C05376=1015.693,102.871,-118.305,166.533,55.921,160.218
C05377=1015.698,103.121,-118.324,166.535,55.912,160.217
C05378=1015.703,103.370,-118.340,166.538,55.902,160.216
C05379=1015.707,103.620,-118.357,166.541,55.892,160.214
C05380=1015.712,103.869,-118.375,166.544,55.882,160.213
C05381=1015.717,104.119,-118.392,166.546,55.872,160.212
C05382=1015.721,104.368,-118.409,166.549,55.862,160.210
C05383=1015.726,104.617,-118.427,166.551,55.852,160.209
C05384=1015.730,104.866,-118.444,166.555,55.842,160.208
C05385=1015.735,105.115,-118.462,166.558,55.832,160.206
C05386=1015.740,105.365,-118.479,166.560,55.822,160.205
C05387=1015.745,105.614,-118.496,166.563,55.812,160.204
C05388=1015.753,106.033,-118.526,166.567,55.795,160.202
C05389=1015.761,106.451,-118.554,166.572,55.778,160.199
C05390=1015.768,106.870,-118.583,166.577,55.761,160.197
C05391=1015.777,107.288,-118.612,166.582,55.744,160.195
C05392=1015.781,107.538,-118.630,166.584,55.735,160.194
C05393=1015.786,107.787,-118.647,166.587,55.724,160.192
C05394=1015.791,108.037,-118.665,166.590,55.714,160.191
C05395=1015.796,108.286,-118.682,166.593,55.704,160.190
C05396=1015.800,108.535,-118.699,166.596,55.694,160.188
C05397=1015.806,108.784,-118.717,166.598,55.684,160.187
C05398=1015.810,109.034,-118.734,166.601,55.673,160.185
C05399=1015.814,109.283,-118.751,166.605,55.664,160.184
C05400=1015.820,109.532,-118.769,166.607,55.654,160.183
C05401=1015.825,109.782,-118.787,166.610,55.644,160.182
C05402=1015.829,110.032,-118.804,166.612,55.634,160.180
C05403=1015.833,110.280,-118.822,166.615,55.623,160.179
C05404=1015.838,110.530,-118.839,166.618,55.614,160.177
C05405=1015.843,110.779,-118.857,166.621,55.604,160.176
C05406=1015.848,111.029,-118.875,166.625,55.594,160.175
C05407=1015.853,111.278,-118.892,166.627,55.584,160.173
C05408=1015.857,111.527,-118.910,166.630,55.573,160.172
C05409=1015.862,111.777,-118.928,166.632,55.564,160.171
C05410=1015.867,112.026,-118.946,166.635,55.554,160.170
C05411=1015.871,112.275,-118.964,166.639,55.544,160.168
C05412=1015.876,112.524,-118.982,166.641,55.534,160.167
C05413=1015.880,112.774,-118.999,166.644,55.525,160.166
C05414=1015.885,113.024,-119.017,166.647,55.514,160.164
C05415=1015.889,113.272,-119.035,166.649,55.505,160.163
C05416=1015.894,113.522,-119.053,166.652,55.495,160.162
C05417=1015.899,113.771,-119.071,166.656,55.485,160.161
C05418=1015.903,114.021,-119.089,166.658,55.475,160.159
C05419=1015.908,114.270,-119.107,166.662,55.465,160.158
C05420=1015.912,114.519,-119.125,166.664,55.455,160.157
C05421=1015.917,114.768,-119.143,166.667,55.445,160.155
C05422=1015.922,115.018,-119.161,166.670,55.435,160.154
C05423=1015.926,115.268,-119.179,166.673,55.425,160.153
C05424=1015.931,115.517,-119.197,166.675,55.416,160.151
C05425=1015.935,115.766,-119.215,166.678,55.405,160.150
C05426=1015.940,116.015,-119.233,166.681,55.396,160.149
C05427=1015.945,116.264,-119.251,166.684,55.386,160.147
C05428=1015.949,116.514,-119.269,166.687,55.376,160.146
C05429=1015.954,116.763,-119.287,166.690,55.366,160.145
C05430=1015.958,117.012,-119.305,166.693,55.356,160.143
C05431=1015.963,117.262,-119.322,166.696,55.346,160.142
C05432=1015.968,117.511,-119.341,166.699,55.336,160.141
C05433=1015.972,117.760,-119.359,166.701,55.327,160.140
C05434=1015.977,118.010,-119.377,166.705,55.316,160.138
C05435=1015.982,118.259,-119.395,166.707,55.307,160.137
C05436=1015.987,118.508,-119.413,166.710,55.297,160.136
C05437=1015.991,118.757,-119.431,166.713,55.286,160.134
C05438=1015.996,119.006,-119.449,166.716,55.277,160.133
C05439=1016.000,119.256,-119.467,166.719,55.266,160.132
C05440=1016.005,119.505,-119.486,166.721,55.256,160.130
C05441=1016.010,119.754,-119.504,166.725,55.247,160.129
C05442=1016.015,120.004,-119.522,166.728,55.236,160.128
C05443=1016.020,120.253,-119.540,166.730,55.226,160.126
C05444=1016.024,120.502,-119.558,166.734,55.217,160.125
C05445=1016.028,120.751,-119.576,166.737,55.206,160.124
C05446=1016.033,121.000,-119.594,166.739,55.196,160.122
C05447=1016.038,121.250,-119.612,166.743,55.187,160.121
C05448=1016.043,121.499,-119.630,166.745,55.177,160.120
C05449=1016.048,121.749,-119.649,166.748,55.166,160.118
C05450=1016.052,121.998,-119.667,166.752,55.157,160.117
C05451=1016.057,122.247,-119.685,166.754,55.147,160.116
C05452=1016.063,122.528,-119.706,166.758,55.135,160.114
C05453=1016.067,122.810,-119.725,166.762,55.124,160.113
C05454=1016.073,123.091,-119.746,166.764,55.113,160.111
C05455=1016.078,123.372,-119.766,166.768,55.101,160.110
C05456=1016.082,123.622,-119.785,166.772,55.092,160.109
C05457=1016.087,123.871,-119.803,166.774,55.082,160.107
C05458=1016.092,124.120,-119.821,166.777,55.071,160.106
C05459=1016.097,124.369,-119.840,166.780,55.061,160.105
C05460=1016.102,124.618,-119.858,166.783,55.052,160.104
C05461=1016.106,124.868,-119.877,166.786,55.042,160.102
C05462=1016.111,125.117,-119.895,166.789,55.031,160.101
C05463=1016.116,125.366,-119.913,166.792,55.021,160.099
C05464=1016.121,125.616,-119.931,166.795,55.012,160.098
C05465=1016.126,125.865,-119.949,166.799,55.001,160.097
C05466=1016.130,126.115,-119.967,166.802,54.991,160.096
C05467=1016.135,126.364,-119.986,166.804,54.981,160.094
C05468=1016.140,126.613,-120.004,166.808,54.971,160.093
C05469=1016.145,126.862,-120.023,166.811,54.961,160.092
C05470=1016.150,127.111,-120.041,166.814,54.951,160.090
C05471=1016.155,127.361,-120.059,166.816,54.941,160.089
C05472=1016.159,127.610,-120.077,166.820,54.930,160.088
C05473=1016.164,127.859,-120.095,166.823,54.921,160.087
C05474=1016.169,128.109,-120.113,166.827,54.911,160.085
C05475=1016.174,128.358,-120.132,166.829,54.901,160.084
C05476=1016.179,128.607,-120.150,166.832,54.890,160.082
C05477=1016.184,128.856,-120.169,166.835,54.880,160.081
C05478=1016.188,129.105,-120.187,166.839,54.870,160.080
C05479=1016.193,129.355,-120.205,166.841,54.860,160.079
C05480=1016.197,129.605,-120.224,166.845,54.850,160.077
C05481=1016.202,129.853,-120.243,166.848,54.840,160.076
C05482=1016.207,130.103,-120.261,166.851,54.831,160.075
C05483=1016.211,130.352,-120.280,166.854,54.820,160.073
C05484=1016.216,130.601,-120.298,166.858,54.811,160.072
C05485=1016.220,130.851,-120.317,166.860,54.801,160.071
C05486=1016.225,131.099,-120.336,166.863,54.791,160.069
C05487=1016.231,131.349,-120.355,166.867,54.781,160.068
C05488=1016.235,131.598,-120.374,166.869,54.771,160.067
C05489=1016.240,131.848,-120.392,166.873,54.761,160.066
C05490=1016.244,132.097,-120.411,166.876,54.751,160.065
C05491=1016.249,132.346,-120.430,166.879,54.741,160.063
C05492=1016.254,132.596,-120.448,166.882,54.731,160.062
C05493=1016.258,132.845,-120.467,166.886,54.721,160.061
C05494=1016.263,133.094,-120.486,166.888,54.712,160.059
C05495=1016.267,133.343,-120.505,166.891,54.701,160.058
C05496=1016.272,133.592,-120.523,166.895,54.692,160.057
C05497=1016.277,133.841,-120.542,166.898,54.681,160.055
C05498=1016.282,134.091,-120.561,166.901,54.672,160.054
C05499=1016.287,134.340,-120.580,166.904,54.662,160.053
C05500=1016.291,134.590,-120.599,166.908,54.652,160.052
C05501=1016.296,134.839,-120.618,166.910,54.642,160.050
C05502=1016.301,135.088,-120.636,166.914,54.632,160.049
C05503=1016.305,135.337,-120.655,166.917,54.622,160.048
C05504=1016.310,135.586,-120.674,166.921,54.612,160.046
C05505=1016.314,135.835,-120.693,166.923,54.602,160.045
C05506=1016.320,136.085,-120.712,166.927,54.592,160.044
C05507=1016.324,136.334,-120.731,166.930,54.582,160.043
C05508=1016.329,136.583,-120.750,166.932,54.572,160.041
C05509=1016.333,136.833,-120.769,166.936,54.563,160.040
C05510=1016.338,137.082,-120.788,166.939,54.552,160.039
C05511=1016.342,137.331,-120.806,166.943,54.542,160.037
C05512=1016.348,137.581,-120.826,166.946,54.533,160.036
C05513=1016.352,137.830,-120.845,166.949,54.523,160.035
C05514=1016.357,138.079,-120.863,166.952,54.512,160.034
C05515=1016.361,138.328,-120.883,166.955,54.503,160.032
C05516=1016.366,138.609,-120.905,166.959,54.492,160.031
C05517=1016.372,138.890,-120.926,166.963,54.481,160.030
C05518=1016.377,139.171,-120.947,166.966,54.470,160.028
C05519=1016.382,139.452,-120.969,166.970,54.458,160.027
C05520=1016.387,139.702,-120.989,166.974,54.449,160.026
C05521=1016.392,139.951,-121.007,166.977,54.439,160.024
C05522=1016.396,140.200,-121.027,166.980,54.429,160.023
C05523=1016.400,140.449,-121.046,166.983,54.419,160.022
C05524=1016.406,140.699,-121.065,166.986,54.409,160.020
C05525=1016.410,140.948,-121.085,166.989,54.400,160.019
C05526=1016.415,141.197,-121.104,166.993,54.390,160.018
C05527=1016.420,141.446,-121.122,166.996,54.379,160.017
C05528=1016.424,141.695,-121.142,167.000,54.370,160.016
C05529=1016.429,141.945,-121.162,167.002,54.360,160.014
C05530=1016.434,142.194,-121.181,167.006,54.350,160.013
C05531=1016.438,142.443,-121.200,167.010,54.340,160.012
C05532=1016.442,142.692,-121.219,167.013,54.330,160.010
C05533=1016.448,142.942,-121.238,167.015,54.320,160.009
C05534=1016.452,143.191,-121.258,167.019,54.311,160.008
C05535=1016.457,143.440,-121.277,167.023,54.301,160.007
C05536=1016.462,143.689,-121.296,167.026,54.290,160.005
C05537=1016.467,143.938,-121.316,167.029,54.281,160.004
C05538=1016.471,144.187,-121.335,167.032,54.271,160.003
C05539=1016.476,144.436,-121.354,167.036,54.261,160.001
C05540=1016.481,144.686,-121.374,167.040,54.251,160.000
C05541=1016.485,144.935,-121.393,167.043,54.241,159.999
C05542=1016.490,145.184,-121.412,167.045,54.231,159.998
C05543=1016.495,145.434,-121.431,167.049,54.222,159.997
C05544=1016.500,145.683,-121.451,167.053,54.212,159.995
C05545=1016.504,145.932,-121.470,167.056,54.202,159.994
C05546=1016.509,146.182,-121.490,167.059,54.192,159.993
C05547=1016.514,146.430,-121.509,167.062,54.182,159.991
C05548=1016.518,146.680,-121.528,167.066,54.173,159.990
C05549=1016.523,146.928,-121.549,167.070,54.163,159.989
C05550=1016.528,147.178,-121.569,167.072,54.153,159.988
C05551=1016.532,147.427,-121.588,167.076,54.143,159.987
C05552=1016.537,147.676,-121.608,167.080,54.133,159.985
C05553=1016.542,147.926,-121.627,167.083,54.124,159.984
C05554=1016.546,148.175,-121.647,167.086,54.114,159.983
C05555=1016.552,148.424,-121.666,167.089,54.104,159.982
C05556=1016.556,148.673,-121.685,167.093,54.094,159.980
C05557=1016.560,148.922,-121.705,167.097,54.084,159.979
C05558=1016.566,149.171,-121.726,167.100,54.075,159.978
C05559=1016.570,149.420,-121.745,167.103,54.065,159.977
C05560=1016.574,149.669,-121.764,167.107,54.055,159.975
C05561=1016.579,149.919,-121.784,167.110,54.045,159.974
C05562=1016.584,150.168,-121.804,167.113,54.035,159.973
C05563=1016.589,150.418,-121.824,167.117,54.026,159.972
C05564=1016.593,150.666,-121.844,167.120,54.016,159.971
C05565=1016.598,150.915,-121.863,167.124,54.006,159.969
C05566=1016.602,151.165,-121.883,167.128,53.996,159.968
C05567=1016.607,151.414,-121.903,167.130,53.986,159.967
C05568=1016.612,151.663,-121.923,167.134,53.977,159.966
C05569=1016.616,151.912,-121.943,167.138,53.967,159.964
C05570=1016.621,152.161,-121.962,167.141,53.957,159.963
C05571=1016.626,152.411,-121.982,167.145,53.947,159.962
C05572=1016.630,152.659,-122.002,167.148,53.938,159.961
C05573=1016.635,152.909,-122.022,167.152,53.928,159.960
C05574=1016.640,153.158,-122.041,167.155,53.918,159.958
C05575=1016.645,153.407,-122.062,167.159,53.908,159.957
C05576=1016.649,153.656,-122.081,167.162,53.898,159.956
C05577=1016.654,153.906,-122.101,167.165,53.889,159.954
C05578=1016.659,154.155,-122.121,167.169,53.879,159.953
C05579=1016.663,154.404,-122.141,167.172,53.869,159.952
C05580=1016.668,154.685,-122.165,167.177,53.858,159.951
C05581=1016.674,154.966,-122.186,167.181,53.847,159.950
C05582=1016.679,155.247,-122.209,167.184,53.837,159.948
C05583=1016.685,155.528,-122.231,167.188,53.825,159.947
C05584=1016.689,155.778,-122.252,167.192,53.815,159.945
C05585=1016.693,156.026,-122.272,167.196,53.806,159.944
C05586=1016.698,156.276,-122.292,167.199,53.796,159.943
C05587=1016.703,156.524,-122.312,167.203,53.786,159.942
C05588=1016.708,156.774,-122.332,167.206,53.777,159.941
C05589=1016.713,157.022,-122.352,167.210,53.767,159.940
C05590=1016.718,157.272,-122.372,167.213,53.757,159.938
C05591=1016.722,157.521,-122.392,167.217,53.747,159.937
C05592=1016.727,157.770,-122.412,167.221,53.738,159.936
C05593=1016.731,158.019,-122.433,167.224,53.727,159.935
C05594=1016.736,158.269,-122.453,167.227,53.718,159.933
C05595=1016.741,158.517,-122.473,167.231,53.708,159.932
C05596=1016.746,158.767,-122.493,167.235,53.699,159.931
C05597=1016.750,159.016,-122.513,167.238,53.689,159.930
C05598=1016.754,159.265,-122.535,167.241,53.680,159.929
C05599=1016.759,159.514,-122.555,167.245,53.670,159.928
C05600=1016.763,159.764,-122.575,167.249,53.660,159.926
C05601=1016.768,160.012,-122.595,167.253,53.651,159.925
C05602=1016.772,160.261,-122.617,167.256,53.642,159.924
C05603=1016.777,160.511,-122.637,167.260,53.632,159.923
C05604=1016.781,160.759,-122.658,167.264,53.623,159.922
C05605=1016.785,161.009,-122.678,167.268,53.613,159.921
C05606=1016.790,161.258,-122.698,167.270,53.603,159.919
C05607=1016.795,161.507,-122.720,167.274,53.594,159.918
C05608=1016.799,161.756,-122.740,167.278,53.584,159.917
C05609=1016.804,162.005,-122.761,167.282,53.575,159.916
C05610=1016.808,162.255,-122.782,167.285,53.566,159.915
C05611=1016.813,162.504,-122.802,167.288,53.556,159.913
C05612=1016.817,162.753,-122.823,167.292,53.546,159.912
C05613=1016.822,163.001,-122.843,167.297,53.537,159.911
C05614=1016.826,163.251,-122.864,167.299,53.527,159.910
C05615=1016.832,163.500,-122.885,167.303,53.518,159.909
C05616=1016.836,163.749,-122.905,167.307,53.508,159.908
C05617=1016.840,163.998,-122.927,167.311,53.498,159.906
C05618=1016.845,164.247,-122.947,167.315,53.489,159.905
C05619=1016.849,164.496,-122.968,167.317,53.479,159.904
C05620=1016.855,164.745,-122.988,167.321,53.470,159.903
C05621=1016.858,164.994,-123.009,167.325,53.460,159.902
C05622=1016.863,165.244,-123.030,167.329,53.451,159.901
C05623=1016.868,165.493,-123.050,167.333,53.441,159.900
C05624=1016.872,165.742,-123.071,167.337,53.431,159.898
C05625=1016.877,165.991,-123.092,167.340,53.422,159.897
C05626=1016.882,166.240,-123.113,167.343,53.412,159.896
C05627=1016.885,166.489,-123.133,167.348,53.403,159.895
C05628=1016.891,166.738,-123.154,167.352,53.394,159.894
C05629=1016.895,166.988,-123.175,167.355,53.384,159.892
C05630=1016.900,167.236,-123.195,167.359,53.374,159.891
C05631=1016.904,167.486,-123.217,167.362,53.365,159.890
C05632=1016.909,167.735,-123.238,167.366,53.355,159.889
C05633=1016.914,167.984,-123.258,167.370,53.346,159.888
C05634=1016.918,168.233,-123.279,167.374,53.336,159.887
C05635=1016.923,168.482,-123.300,167.378,53.327,159.886
C05636=1016.928,168.731,-123.321,167.381,53.317,159.884
C05637=1016.932,168.979,-123.342,167.386,53.307,159.883
C05638=1016.937,169.229,-123.363,167.390,53.298,159.882
C05639=1016.942,169.478,-123.384,167.393,53.288,159.881
C05640=1016.947,169.727,-123.404,167.396,53.279,159.880
C05641=1016.951,169.976,-123.425,167.400,53.269,159.878
C05642=1016.956,170.225,-123.446,167.404,53.260,159.877
C05643=1016.961,170.474,-123.467,167.408,53.250,159.876
C05644=1016.966,170.755,-123.491,167.412,53.239,159.875
C05645=1016.971,171.036,-123.515,167.417,53.228,159.874
C05646=1016.977,171.317,-123.538,167.421,53.218,159.872
C05647=1016.983,171.597,-123.562,167.426,53.207,159.871
C05648=1016.986,171.846,-123.583,167.429,53.197,159.870
C05649=1016.992,172.095,-123.603,167.433,53.187,159.869
C05650=1016.996,172.345,-123.624,167.438,53.178,159.868
C05651=1017.001,172.594,-123.646,167.441,53.168,159.866
C05652=1017.006,172.843,-123.666,167.445,53.159,159.865
C05653=1017.011,173.092,-123.688,167.449,53.149,159.864
C05654=1017.015,173.340,-123.708,167.453,53.140,159.863
C05655=1017.020,173.590,-123.729,167.457,53.130,159.862
C05656=1017.024,173.839,-123.750,167.461,53.120,159.861
C05657=1017.030,174.088,-123.772,167.465,53.110,159.859
C05658=1017.035,174.337,-123.793,167.469,53.101,159.858
C05659=1017.039,174.587,-123.814,167.473,53.092,159.857
C05660=1017.044,174.836,-123.835,167.477,53.082,159.856
C05661=1017.049,175.084,-123.856,167.481,53.073,159.855
C05662=1017.054,175.333,-123.877,167.484,53.063,159.854
C05663=1017.058,175.582,-123.898,167.489,53.053,159.853
C05664=1017.063,175.831,-123.920,167.492,53.043,159.851
C05665=1017.068,176.080,-123.940,167.496,53.034,159.850
C05666=1017.073,176.330,-123.961,167.500,53.024,159.849
C05667=1017.078,176.579,-123.982,167.504,53.015,159.848
C05668=1017.083,176.828,-124.004,167.508,53.006,159.847
C05669=1017.088,177.077,-124.025,167.512,52.996,159.846
C05670=1017.093,177.326,-124.046,167.516,52.986,159.845
C05671=1017.098,177.575,-124.067,167.520,52.976,159.843
C05672=1017.102,177.825,-124.088,167.524,52.967,159.842
C05673=1017.108,178.073,-124.110,167.528,52.957,159.841
C05674=1017.112,178.323,-124.131,167.532,52.948,159.840
C05675=1017.117,178.571,-124.151,167.536,52.938,159.839
C05676=1017.122,178.820,-124.173,167.540,52.929,159.838
C05677=1017.126,179.069,-124.194,167.544,52.919,159.837
C05678=1017.132,179.318,-124.215,167.548,52.910,159.835
C05679=1017.136,179.567,-124.236,167.553,52.899,159.834
C05680=1017.141,179.816,-124.258,167.557,52.890,159.833
C05681=1017.146,180.065,-124.279,167.561,52.881,159.832
C05682=1017.151,180.315,-124.300,167.565,52.871,159.831
C05683=1017.156,180.563,-124.321,167.569,52.862,159.830
C05684=1017.161,180.812,-124.342,167.573,52.852,159.829
C05685=1017.166,181.062,-124.365,167.577,52.843,159.828
C05686=1017.172,181.311,-124.385,167.581,52.833,159.826
C05687=1017.176,181.560,-124.407,167.585,52.823,159.825
C05688=1017.181,181.809,-124.428,167.590,52.813,159.824
C05689=1017.186,182.058,-124.450,167.594,52.804,159.823
C05690=1017.191,182.307,-124.472,167.597,52.795,159.822
C05691=1017.195,182.556,-124.494,167.601,52.786,159.821
C05692=1017.199,182.806,-124.516,167.605,52.777,159.820
C05693=1017.204,183.054,-124.537,167.610,52.767,159.819
C05694=1017.209,183.303,-124.559,167.614,52.758,159.818
C05695=1017.213,183.552,-124.582,167.618,52.749,159.817
C05696=1017.218,183.801,-124.604,167.622,52.739,159.815
C05697=1017.223,184.050,-124.625,167.626,52.730,159.814
C05698=1017.227,184.299,-124.647,167.630,52.721,159.813
C05699=1017.232,184.548,-124.670,167.635,52.711,159.812
C05700=1017.236,184.797,-124.692,167.639,52.702,159.811
C05701=1017.241,185.045,-124.714,167.643,52.693,159.810
C05702=1017.245,185.295,-124.735,167.647,52.684,159.809
C05703=1017.250,185.544,-124.757,167.651,52.675,159.808
C05704=1017.255,185.794,-124.779,167.655,52.665,159.807
C05705=1017.260,186.042,-124.801,167.659,52.656,159.806
C05706=1017.264,186.292,-124.824,167.664,52.646,159.805
C05707=1017.269,186.540,-124.846,167.668,52.637,159.804
C05708=1017.275,186.820,-124.871,167.673,52.627,159.803
C05709=1017.280,187.101,-124.896,167.677,52.616,159.801
C05710=1017.285,187.381,-124.920,167.682,52.606,159.800
C05711=1017.290,187.662,-124.945,167.687,52.596,159.799
C05712=1017.294,187.910,-124.967,167.691,52.586,159.798
C05713=1017.300,188.160,-124.989,167.695,52.577,159.797
C05714=1017.304,188.409,-125.012,167.699,52.568,159.796
C05715=1017.309,188.658,-125.034,167.703,52.558,159.795
C05716=1017.314,188.906,-125.056,167.708,52.549,159.794
C05717=1017.319,189.155,-125.078,167.712,52.540,159.792
C05718=1017.323,189.404,-125.100,167.716,52.531,159.791
C05719=1017.328,189.654,-125.123,167.721,52.521,159.791
C05720=1017.333,189.902,-125.145,167.726,52.512,159.789
C05721=1017.337,190.152,-125.167,167.730,52.503,159.788
C05722=1017.342,190.400,-125.189,167.734,52.494,159.787
C05723=1017.347,190.649,-125.211,167.738,52.484,159.786
C05724=1017.352,190.899,-125.233,167.742,52.475,159.785
C05725=1017.357,191.147,-125.256,167.746,52.465,159.784
C05726=1017.361,191.396,-125.278,167.751,52.456,159.783
C05727=1017.366,191.645,-125.300,167.755,52.447,159.782
C05728=1017.371,191.895,-125.323,167.759,52.438,159.781
C05729=1017.376,192.143,-125.345,167.765,52.429,159.780
C05730=1017.381,192.392,-125.367,167.769,52.419,159.779
C05731=1017.386,192.640,-125.389,167.773,52.410,159.778
C05732=1017.390,192.890,-125.412,167.777,52.400,159.777
C05733=1017.395,193.139,-125.434,167.781,52.391,159.776
C05734=1017.400,193.387,-125.456,167.786,52.382,159.775
C05735=1017.405,193.637,-125.479,167.790,52.373,159.774
C05736=1017.410,193.886,-125.501,167.795,52.364,159.773
C05737=1017.415,194.135,-125.523,167.799,52.354,159.772
C05738=1017.419,194.383,-125.546,167.804,52.345,159.771
C05739=1017.424,194.633,-125.568,167.808,52.335,159.769
C05740=1017.429,194.882,-125.590,167.812,52.326,159.768
C05741=1017.434,195.130,-125.613,167.816,52.317,159.767
C05742=1017.439,195.380,-125.636,167.822,52.308,159.766
C05743=1017.444,195.628,-125.657,167.826,52.299,159.765
C05744=1017.450,195.877,-125.680,167.830,52.289,159.764
C05745=1017.454,196.126,-125.703,167.834,52.280,159.763
C05746=1017.459,196.375,-125.725,167.839,52.271,159.762
C05747=1017.464,196.624,-125.748,167.844,52.262,159.761
C05748=1017.468,196.873,-125.770,167.848,52.253,159.760
C05749=1017.474,197.121,-125.793,167.852,52.243,159.759
C05750=1017.479,197.371,-125.815,167.857,52.234,159.758
C05751=1017.483,197.620,-125.837,167.862,52.224,159.757
C05752=1017.489,197.869,-125.860,167.866,52.215,159.756
C05753=1017.494,198.118,-125.882,167.871,52.206,159.755
C05754=1017.499,198.367,-125.905,167.875,52.197,159.754
C05755=1017.503,198.616,-125.928,167.880,52.188,159.753
C05756=1017.509,198.864,-125.950,167.885,52.178,159.752
C05757=1017.514,199.114,-125.972,167.889,52.169,159.751
C05758=1017.518,199.362,-125.996,167.893,52.160,159.750
C05759=1017.523,199.612,-126.018,167.899,52.151,159.749
C05760=1017.528,199.860,-126.041,167.903,52.142,159.748
C05761=1017.533,200.109,-126.064,167.907,52.133,159.747
C05762=1017.537,200.358,-126.087,167.912,52.124,159.746
C05763=1017.543,200.607,-126.110,167.916,52.114,159.745
C05764=1017.547,200.856,-126.133,167.920,52.105,159.744
C05765=1017.552,201.104,-126.156,167.926,52.096,159.743
C05766=1017.557,201.354,-126.178,167.930,52.087,159.742
C05767=1017.562,201.602,-126.202,167.935,52.078,159.741
C05768=1017.567,201.852,-126.225,167.939,52.069,159.740
C05769=1017.572,202.100,-126.248,167.943,52.060,159.739
C05770=1017.577,202.349,-126.271,167.949,52.051,159.738
C05771=1017.600,203.593,-126.387,168.432,52.137,159.849
C05772=1017.606,203.828,-126.409,168.436,52.129,159.848
C05773=1017.612,204.063,-126.433,168.440,52.122,159.847
C05774=1017.618,204.298,-126.456,168.443,52.114,159.846
C05775=1017.623,204.534,-126.479,168.447,52.107,159.845
C05776=1017.629,204.769,-126.502,168.450,52.099,159.844
C05777=1017.634,205.003,-126.526,168.454,52.091,159.844
C05778=1017.640,205.238,-126.549,168.458,52.084,159.843
C05779=1017.645,205.473,-126.572,168.462,52.076,159.842
C05780=1017.651,205.722,-126.598,168.466,52.068,159.841
C05781=1017.657,205.970,-126.622,168.470,52.061,159.840
C05782=1017.663,206.219,-126.647,168.474,52.053,159.839
C05783=1017.669,206.468,-126.672,168.477,52.045,159.838
C05784=1017.674,206.716,-126.697,168.481,52.037,159.837
C05785=1017.680,206.966,-126.721,168.485,52.030,159.836
C05786=1017.686,207.214,-126.746,168.490,52.021,159.835
C05787=1017.692,207.463,-126.771,168.494,52.013,159.834
C05788=1017.698,207.712,-126.796,168.498,52.006,159.834
C05789=1017.703,207.960,-126.821,168.501,51.998,159.833
C05790=1017.709,208.209,-126.846,168.505,51.990,159.832
C05791=1017.716,208.458,-126.871,168.509,51.983,159.831
C05792=1017.721,208.706,-126.896,168.513,51.975,159.830
C05793=1017.727,208.955,-126.921,168.517,51.967,159.829
C05794=1017.732,209.204,-126.946,168.521,51.960,159.828
C05795=1017.738,209.452,-126.971,168.525,51.951,159.827
C05796=1017.744,209.701,-126.996,168.530,51.944,159.826
C05797=1017.750,209.950,-127.022,168.533,51.936,159.825
C05798=1017.756,210.198,-127.046,168.537,51.929,159.825
C05799=1017.762,210.447,-127.071,168.541,51.921,159.824
C05800=1017.767,210.696,-127.097,168.545,51.913,159.823
C05801=1017.773,210.944,-127.122,168.549,51.905,159.822
C05802=1017.779,211.193,-127.147,168.553,51.898,159.821
C05803=1017.785,211.442,-127.172,168.557,51.890,159.820
C05804=1017.790,211.690,-127.198,168.561,51.883,159.819
C05805=1017.796,211.939,-127.223,168.565,51.876,159.818
C05806=1017.802,212.187,-127.248,168.569,51.868,159.817
C05807=1017.808,212.436,-127.274,168.573,51.860,159.817
C05808=1017.813,212.685,-127.299,168.577,51.853,159.816
C05809=1017.819,212.934,-127.324,168.581,51.845,159.815
C05810=1017.825,213.182,-127.349,168.585,51.838,159.814
C05811=1017.831,213.431,-127.375,168.589,51.830,159.813
C05812=1017.836,213.679,-127.400,168.593,51.823,159.812
C05813=1017.843,213.928,-127.426,168.597,51.816,159.811
C05814=1017.849,214.177,-127.451,168.601,51.808,159.810
C05815=1017.854,214.426,-127.477,168.605,51.800,159.810
C05816=1017.860,214.674,-127.501,168.609,51.793,159.809
C05817=1017.866,214.923,-127.526,168.613,51.786,159.808
C05818=1017.871,215.172,-127.552,168.617,51.778,159.807
C05819=1017.878,215.421,-127.578,168.621,51.771,159.806
C05820=1017.884,215.669,-127.603,168.625,51.763,159.806
C05821=1017.889,215.917,-127.628,168.630,51.756,159.805
C05822=1017.895,216.166,-127.654,168.633,51.748,159.804
C05823=1017.901,216.415,-127.679,168.636,51.741,159.803
C05824=1017.907,216.663,-127.705,168.641,51.734,159.802
C05825=1017.913,216.912,-127.730,168.645,51.727,159.801
C05826=1017.919,217.161,-127.756,168.648,51.719,159.800
C05827=1017.925,217.410,-127.781,168.653,51.712,159.799
C05828=1017.931,217.658,-127.806,168.657,51.704,159.799
C05829=1017.937,217.906,-127.832,168.661,51.697,159.798
C05830=1017.943,218.155,-127.858,168.665,51.690,159.797
C05831=1017.949,218.403,-127.884,168.669,51.683,159.796
C05832=1017.959,218.817,-127.926,168.675,51.671,159.795
C05833=1017.966,219.179,-127.964,168.681,51.660,159.794
C05834=1017.975,219.540,-128.002,168.687,51.650,159.793
C05835=1017.983,219.901,-128.039,168.693,51.640,159.792
C05836=1017.992,220.263,-128.077,168.699,51.629,159.790
C05837=1017.998,220.512,-128.103,168.704,51.622,159.790
C05838=1018.003,220.760,-128.128,168.708,51.615,159.789
C05839=1018.009,221.009,-128.154,168.712,51.608,159.788
C05840=1018.015,221.257,-128.180,168.716,51.600,159.787
C05841=1018.021,221.506,-128.206,168.719,51.594,159.786
C05842=1018.026,221.755,-128.232,168.723,51.586,159.786
C05843=1018.033,222.003,-128.258,168.728,51.580,159.785
C05844=1018.038,222.252,-128.284,168.732,51.573,159.784
C05845=1018.044,222.500,-128.309,168.736,51.565,159.783
C05846=1018.050,222.749,-128.336,168.741,51.558,159.783
C05847=1018.056,222.997,-128.361,168.744,51.551,159.782
C05848=1018.062,223.246,-128.387,168.748,51.544,159.781
C05849=1018.068,223.495,-128.413,168.753,51.537,159.780
C05850=1018.074,223.743,-128.439,168.757,51.530,159.780
C05851=1018.080,223.992,-128.465,168.761,51.523,159.779
C05852=1018.086,224.240,-128.491,168.765,51.516,159.778
C05853=1018.091,224.489,-128.517,168.769,51.510,159.777
C05854=1018.097,224.738,-128.543,168.773,51.502,159.777
C05855=1018.103,224.986,-128.569,168.777,51.495,159.776
C05856=1018.109,225.235,-128.595,168.781,51.488,159.775
C05857=1018.115,225.483,-128.621,168.786,51.482,159.774
C05858=1018.121,225.732,-128.647,168.789,51.475,159.774
C05859=1018.127,225.980,-128.673,168.793,51.467,159.773
C05860=1018.133,226.229,-128.699,168.798,51.461,159.772
C05861=1018.138,226.478,-128.725,168.802,51.454,159.771
C05862=1018.145,226.726,-128.751,168.806,51.447,159.771
C05863=1018.151,226.974,-128.778,168.810,51.440,159.770
C05864=1018.156,227.223,-128.804,168.814,51.433,159.769
C05865=1018.162,227.471,-128.831,168.819,51.427,159.769
C05866=1018.168,227.720,-128.858,168.822,51.420,159.768
C05867=1018.174,227.969,-128.883,168.827,51.413,159.767
C05868=1018.180,228.218,-128.910,168.831,51.406,159.766
C05869=1018.186,228.466,-128.936,168.836,51.400,159.766
C05870=1018.191,228.715,-128.962,168.839,51.393,159.765
C05871=1018.197,228.963,-128.989,168.843,51.386,159.764
C05872=1018.203,229.212,-129.015,168.848,51.379,159.764
C05873=1018.209,229.460,-129.042,168.851,51.373,159.763
C05874=1018.215,229.709,-129.067,168.856,51.366,159.762
C05875=1018.221,229.957,-129.094,168.860,51.359,159.762
C05876=1018.227,230.205,-129.121,168.865,51.353,159.761
C05877=1018.233,230.454,-129.148,168.868,51.347,159.760
C05878=1018.239,230.703,-129.174,168.873,51.339,159.759
C05879=1018.244,230.951,-129.201,168.877,51.333,159.759
C05880=1018.250,231.199,-129.228,168.881,51.327,159.758
C05881=1018.256,231.448,-129.254,168.885,51.320,159.757
C05882=1018.262,231.697,-129.280,168.890,51.313,159.757
C05883=1018.267,231.945,-129.307,168.893,51.307,159.756
C05884=1018.274,232.194,-129.334,168.898,51.300,159.755
C05885=1018.279,232.443,-129.361,168.902,51.293,159.755
C05886=1018.285,232.691,-129.387,168.906,51.287,159.754
C05887=1018.291,232.939,-129.414,168.911,51.281,159.754
C05888=1018.297,233.188,-129.441,168.914,51.275,159.753
C05889=1018.302,233.416,-129.465,168.919,51.268,159.752
C05890=1018.308,233.644,-129.490,168.922,51.262,159.752
C05891=1018.313,233.872,-129.514,168.926,51.256,159.751
C05892=1018.318,234.101,-129.539,168.930,51.250,159.750
C05893=1018.324,234.329,-129.563,168.934,51.244,159.750
C05894=1018.330,234.558,-129.588,168.937,51.238,159.749
C05895=1018.334,234.786,-129.613,168.941,51.233,159.749
C05896=1018.341,235.014,-129.637,168.945,51.226,159.748
C05897=1018.346,235.262,-129.663,168.950,51.220,159.747
C05898=1018.353,235.511,-129.690,168.954,51.213,159.747
C05899=1018.358,235.760,-129.717,168.958,51.207,159.746
C05900=1018.365,236.007,-129.744,168.963,51.201,159.746
C05901=1018.370,236.256,-129.771,168.966,51.195,159.745
C05902=1018.377,236.505,-129.798,168.971,51.188,159.744
C05903=1018.382,236.753,-129.825,168.976,51.182,159.744
C05904=1018.387,237.002,-129.852,168.979,51.176,159.743
C05905=1018.393,237.250,-129.879,168.984,51.169,159.743
C05906=1018.400,237.499,-129.906,168.988,51.162,159.742
C05907=1018.406,237.747,-129.933,168.992,51.156,159.741
C05908=1018.412,237.995,-129.960,168.997,51.150,159.741
C05909=1018.418,238.244,-129.987,169.000,51.144,159.740
C05910=1018.424,238.493,-130.013,169.005,51.138,159.739
C05911=1018.429,238.741,-130.040,169.010,51.131,159.739
C05912=1018.436,238.990,-130.068,169.013,51.125,159.738
C05913=1018.442,239.238,-130.094,169.018,51.118,159.738
C05914=1018.447,239.487,-130.122,169.022,51.112,159.737
C05915=1018.454,239.735,-130.149,169.026,51.106,159.736
C05916=1018.459,239.983,-130.176,169.030,51.100,159.736
C05917=1018.465,240.231,-130.204,169.035,51.094,159.735
C05918=1018.471,240.481,-130.231,169.039,51.088,159.735
C05919=1018.477,240.729,-130.258,169.043,51.081,159.734
C05920=1018.483,240.978,-130.286,169.047,51.075,159.733
C05921=1018.489,241.226,-130.313,169.052,51.070,159.733
C05922=1018.495,241.474,-130.340,169.056,51.063,159.732
C05923=1018.500,241.723,-130.368,169.061,51.057,159.732
C05924=1018.506,241.971,-130.395,169.064,51.051,159.731
C05925=1018.513,242.220,-130.422,169.069,51.045,159.731
C05926=1018.518,242.468,-130.450,169.074,51.039,159.730
C05927=1018.524,242.716,-130.477,169.078,51.033,159.729
C05928=1018.531,242.965,-130.504,169.083,51.027,159.729
C05929=1018.536,243.213,-130.532,169.086,51.021,159.728
C05930=1018.542,243.462,-130.559,169.091,51.015,159.728
C05931=1018.548,243.710,-130.587,169.095,51.009,159.727
C05932=1018.553,243.958,-130.615,169.099,51.003,159.727
C05933=1018.559,244.207,-130.642,169.104,50.997,159.726
C05934=1018.565,244.455,-130.670,169.107,50.991,159.726
C05935=1018.571,244.704,-130.698,169.113,50.985,159.725
C05936=1018.576,244.952,-130.725,169.117,50.980,159.725
C05937=1018.582,245.201,-130.753,169.121,50.973,159.724
C05938=1018.588,245.449,-130.781,169.125,50.968,159.724
C05939=1018.594,245.697,-130.809,169.130,50.961,159.723
C05940=1018.600,245.945,-130.837,169.134,50.956,159.723
C05941=1018.606,246.195,-130.864,169.138,50.950,159.722
C05942=1018.611,246.443,-130.892,169.143,50.944,159.722
C05943=1018.617,246.691,-130.920,169.147,50.939,159.721
C05944=1018.623,246.939,-130.948,169.152,50.932,159.720
C05945=1018.629,247.188,-130.976,169.156,50.927,159.720
C05946=1018.635,247.436,-131.003,169.160,50.920,159.719
C05947=1018.641,247.685,-131.031,169.164,50.915,159.719
C05948=1018.646,247.933,-131.059,169.169,50.910,159.718
C05949=1018.652,248.158,-131.085,169.173,50.904,159.718
C05950=1018.657,248.383,-131.109,169.177,50.899,159.718
C05951=1018.663,248.608,-131.135,169.181,50.893,159.717
C05952=1018.668,248.833,-131.160,169.185,50.888,159.717
C05953=1018.674,249.058,-131.185,169.189,50.883,159.716
C05954=1018.679,249.283,-131.210,169.192,50.878,159.716
C05955=1018.684,249.507,-131.235,169.196,50.873,159.715
C05956=1018.689,249.733,-131.262,169.201,50.867,159.715
C05957=1018.696,249.981,-131.289,169.205,50.862,159.714
C05958=1018.701,250.229,-131.317,169.210,50.856,159.714
C05959=1018.708,250.478,-131.345,169.214,50.851,159.714
C05960=1018.714,250.726,-131.373,169.218,50.844,159.713
C05961=1018.719,250.974,-131.401,169.223,50.839,159.712
C05962=1018.726,251.223,-131.429,169.228,50.833,159.712
C05963=1018.731,251.471,-131.457,169.232,50.828,159.712
C05964=1018.737,251.720,-131.485,169.236,50.822,159.711
C05965=1018.744,251.968,-131.513,169.240,50.816,159.711
C05966=1018.749,252.216,-131.541,169.245,50.811,159.710
C05967=1018.755,252.465,-131.569,169.250,50.805,159.710
C05968=1018.762,252.713,-131.597,169.254,50.799,159.709
C05969=1018.767,252.961,-131.625,169.259,50.794,159.709
C05970=1018.773,253.210,-131.653,169.263,50.788,159.708
C05971=1018.780,253.459,-131.681,169.267,50.783,159.708
C05972=1018.786,253.706,-131.710,169.272,50.777,159.707
C05973=1018.792,253.954,-131.738,169.276,50.771,159.707
C05974=1018.798,254.203,-131.766,169.281,50.765,159.706
C05975=1018.804,254.452,-131.794,169.285,50.760,159.706
C05976=1018.810,254.700,-131.822,169.290,50.754,159.706
C05977=1018.816,254.948,-131.850,169.294,50.749,159.705
C05978=1018.823,255.197,-131.879,169.298,50.744,159.705
C05979=1018.829,255.445,-131.907,169.303,50.738,159.704
C05980=1018.835,255.693,-131.935,169.307,50.732,159.704
C05981=1018.840,255.942,-131.963,169.313,50.727,159.703
C05982=1018.847,256.190,-131.991,169.317,50.721,159.703
C05983=1018.853,256.438,-132.020,169.322,50.716,159.703
C05984=1018.859,256.687,-132.048,169.326,50.710,159.702
C05985=1018.865,256.935,-132.075,169.330,50.705,159.702
C05986=1018.872,257.183,-132.104,169.335,50.699,159.701
C05987=1018.878,257.432,-132.133,169.339,50.694,159.701
C05988=1018.884,257.680,-132.161,169.344,50.688,159.700
C05989=1018.891,257.928,-132.190,169.348,50.683,159.700
C05990=1018.896,258.177,-132.218,169.352,50.677,159.699
C05991=1018.903,258.425,-132.245,169.358,50.672,159.699
C05992=1018.909,258.673,-132.274,169.362,50.667,159.699
C05993=1018.915,258.922,-132.303,169.367,50.661,159.698
C05994=1018.922,259.170,-132.331,169.371,50.656,159.698
C05995=1018.928,259.418,-132.359,169.376,50.650,159.697
C05996=1018.934,259.667,-132.388,169.380,50.645,159.697
C05997=1018.941,259.915,-132.416,169.385,50.639,159.697
C05998=1018.946,260.162,-132.445,169.390,50.634,159.696
C05999=1018.952,260.411,-132.473,169.394,50.629,159.696
C06000=1018.958,260.659,-132.502,169.398,50.624,159.695
C06001=1018.965,260.907,-132.531,169.404,50.618,159.695
C06002=1018.971,261.156,-132.560,169.408,50.613,159.695
C06003=1018.976,261.404,-132.589,169.412,50.608,159.694
C06004=1018.982,261.653,-132.618,169.417,50.603,159.694
C06005=1018.988,261.901,-132.647,169.422,50.597,159.694
C06006=1018.995,262.149,-132.676,169.426,50.593,159.693
C06007=1019.000,262.397,-132.704,169.431,50.587,159.693
C06008=1019.007,262.645,-132.733,169.436,50.582,159.693
C06009=1019.012,262.870,-132.759,169.440,50.578,159.692
C06010=1019.018,263.094,-132.785,169.444,50.573,159.692
C06011=1019.023,263.318,-132.812,169.448,50.569,159.692
C06012=1019.028,263.542,-132.837,169.453,50.564,159.691
C06013=1019.034,263.766,-132.863,169.457,50.558,159.691
C06014=1019.040,263.990,-132.890,169.460,50.554,159.691
C06015=1019.045,264.214,-132.916,169.465,50.549,159.690
C06016=1019.051,264.439,-132.942,169.469,50.545,159.690
C06017=1019.057,264.687,-132.971,169.474,50.540,159.690
C06018=1019.063,264.936,-133.000,169.478,50.535,159.689
C06019=1019.069,265.184,-133.029,169.483,50.530,159.689
C06020=1019.076,265.432,-133.058,169.488,50.525,159.689
C06021=1019.082,265.680,-133.087,169.492,50.520,159.688
C06022=1019.087,265.928,-133.117,169.496,50.515,159.688
C06023=1019.094,266.176,-133.146,169.502,50.510,159.688
C06024=1019.100,266.425,-133.175,169.506,50.505,159.687
C06025=1019.106,266.673,-133.204,169.511,50.500,159.687
C06026=1019.112,266.921,-133.234,169.516,50.495,159.687
C06027=1019.118,267.169,-133.263,169.520,50.490,159.686
C06028=1019.124,267.417,-133.292,169.525,50.485,159.686
C06029=1019.130,267.666,-133.321,169.530,50.480,159.686
C06030=1019.136,267.914,-133.350,169.535,50.475,159.686
C06031=1019.142,268.162,-133.379,169.539,50.470,159.685
C06032=1019.149,268.410,-133.409,169.543,50.465,159.685
C06033=1019.155,268.658,-133.438,169.549,50.460,159.685
C06034=1019.161,268.906,-133.468,169.553,50.455,159.685
C06035=1019.167,269.154,-133.497,169.558,50.451,159.684
C06036=1019.173,269.403,-133.526,169.563,50.445,159.684
C06037=1019.179,269.651,-133.555,169.568,50.440,159.684
C06038=1019.186,269.899,-133.586,169.572,50.436,159.683
C06039=1019.192,270.147,-133.615,169.577,50.431,159.683
C06040=1019.197,270.396,-133.644,169.582,50.426,159.683
C06041=1019.204,270.643,-133.674,169.587,50.421,159.683
C06042=1019.209,270.892,-133.704,169.591,50.417,159.682
C06043=1019.216,271.140,-133.733,169.596,50.412,159.682
C06044=1019.222,271.387,-133.763,169.601,50.407,159.682
C06045=1019.228,271.636,-133.793,169.606,50.402,159.682
C06046=1019.235,271.885,-133.822,169.610,50.398,159.681
C06047=1019.240,272.132,-133.852,169.615,50.393,159.681
C06048=1019.247,272.381,-133.881,169.620,50.388,159.681
C06049=1019.252,272.629,-133.911,169.625,50.383,159.681
C06050=1019.259,272.877,-133.941,169.629,50.379,159.680
C06051=1019.265,273.126,-133.970,169.634,50.374,159.680
C06052=1019.271,273.373,-134.000,169.639,50.369,159.680
C06053=1019.277,273.622,-134.030,169.644,50.364,159.679
C06054=1019.284,273.869,-134.059,169.648,50.360,159.679
C06055=1019.290,274.118,-134.089,169.653,50.355,159.679
C06056=1019.296,274.366,-134.119,169.659,50.351,159.679
C06057=1019.302,274.614,-134.149,169.663,50.346,159.679
C06058=1019.308,274.862,-134.179,169.668,50.341,159.678
C06059=1019.315,275.110,-134.209,169.672,50.337,159.678
C06060=1019.321,275.358,-134.238,169.678,50.332,159.678
C06061=1019.327,275.606,-134.269,169.683,50.328,159.678
C06062=1019.334,275.855,-134.298,169.687,50.323,159.678
C06063=1019.339,276.103,-134.329,169.692,50.318,159.677
C06064=1019.346,276.350,-134.358,169.697,50.313,159.677
C06065=1019.351,276.599,-134.388,169.702,50.309,159.677
C06066=1019.359,276.847,-134.418,169.707,50.305,159.677
C06067=1019.364,277.095,-134.448,169.711,50.300,159.676
C06068=1019.370,277.343,-134.479,169.717,50.295,159.676
C06069=1019.376,277.570,-134.506,169.720,50.291,159.676
C06070=1019.382,277.796,-134.533,169.725,50.287,159.676
C06071=1019.387,278.022,-134.561,169.730,50.283,159.676
C06072=1019.393,278.249,-134.589,169.734,50.279,159.676
C06073=1019.398,278.475,-134.617,169.739,50.275,159.675
C06074=1019.404,278.701,-134.644,169.744,50.271,159.675
C06075=1019.410,278.928,-134.671,169.747,50.267,159.675
C06076=1019.415,279.154,-134.699,169.752,50.263,159.675
C06077=1019.422,279.403,-134.730,169.757,50.259,159.675
C06078=1019.428,279.650,-134.760,169.761,50.254,159.675
C06079=1019.435,279.899,-134.791,169.767,50.250,159.675
C06080=1019.440,280.147,-134.820,169.772,50.245,159.674
C06081=1019.446,280.395,-134.850,169.777,50.241,159.674
C06082=1019.452,280.643,-134.881,169.781,50.237,159.674
C06083=1019.459,280.891,-134.911,169.787,50.232,159.674
C06084=1019.465,281.139,-134.942,169.792,50.228,159.674
C06085=1019.471,281.387,-134.972,169.797,50.224,159.674
C06086=1019.477,281.636,-135.003,169.801,50.220,159.673
C06087=1019.484,281.883,-135.033,169.806,50.215,159.673
C06088=1019.491,282.131,-135.064,169.812,50.211,159.673
C06089=1019.497,282.379,-135.094,169.816,50.206,159.673
C06090=1019.502,282.627,-135.125,169.821,50.202,159.673
C06091=1019.509,282.875,-135.155,169.826,50.198,159.673
C06092=1019.515,283.123,-135.185,169.832,50.193,159.673
C06093=1019.522,283.371,-135.216,169.837,50.189,159.672
C06094=1019.528,283.620,-135.247,169.842,50.185,159.672
C06095=1019.534,283.868,-135.277,169.846,50.180,159.672
C06096=1019.541,284.115,-135.308,169.852,50.176,159.672
C06097=1019.547,284.363,-135.338,169.857,50.172,159.672
C06098=1019.554,284.612,-135.369,169.861,50.168,159.672
C06099=1019.560,284.859,-135.399,169.866,50.164,159.672
C06100=1019.566,285.107,-135.431,169.871,50.160,159.672
C06101=1019.572,285.355,-135.461,169.877,50.155,159.672
C06102=1019.578,285.604,-135.492,169.882,50.151,159.671
C06103=1019.585,285.851,-135.523,169.887,50.147,159.671
C06104=1019.591,286.099,-135.553,169.891,50.143,159.671
C06105=1019.597,286.348,-135.584,169.896,50.139,159.671
C06106=1019.604,286.595,-135.615,169.902,50.134,159.671
C06107=1019.610,286.844,-135.646,169.907,50.130,159.671
C06108=1019.616,287.091,-135.677,169.912,50.126,159.671
C06109=1019.623,287.339,-135.708,169.917,50.123,159.671
C06110=1019.629,287.587,-135.739,169.923,50.118,159.671
C06111=1019.635,287.835,-135.770,169.928,50.114,159.671
C06112=1019.642,288.083,-135.801,169.933,50.110,159.671
C06113=1019.648,288.332,-135.832,169.938,50.106,159.670
C06114=1019.654,288.579,-135.863,169.943,50.102,159.670
C06115=1019.661,288.827,-135.893,169.948,50.098,159.670
C06116=1019.667,289.075,-135.925,169.953,50.094,159.670
C06117=1019.673,289.323,-135.955,169.958,50.090,159.670
C06118=1019.680,289.571,-135.987,169.963,50.086,159.670
C06119=1019.687,289.819,-136.018,169.968,50.082,159.670
C06120=1019.693,290.067,-136.048,169.974,50.078,159.670
C06121=1019.699,290.315,-136.080,169.979,50.074,159.670
C06122=1019.705,290.563,-136.112,169.984,50.070,159.670
C06123=1019.711,290.811,-136.142,169.989,50.066,159.670
C06124=1019.718,291.058,-136.174,169.994,50.062,159.670
C06125=1019.725,291.306,-136.205,170.000,50.058,159.670
C06126=1019.731,291.554,-136.237,170.005,50.054,159.670
C06127=1019.737,291.802,-136.267,170.010,50.050,159.670
C06128=1019.743,292.050,-136.299,170.015,50.046,159.670
C06129=1019.750,292.283,-136.328,170.020,50.043,159.670
C06130=1019.755,292.516,-136.358,170.025,50.039,159.670
C06131=1019.762,292.748,-136.387,170.030,50.036,159.670
C06132=1019.767,292.981,-136.417,170.035,50.032,159.670
C06133=1019.774,293.213,-136.446,170.039,50.028,159.669
C06134=1019.779,293.446,-136.476,170.044,50.025,159.670
C06135=1019.785,293.678,-136.505,170.050,50.022,159.670
C06136=1019.791,293.910,-136.536,170.054,50.018,159.670
C06137=1019.797,294.158,-136.567,170.060,50.014,159.670
C06138=1019.803,294.406,-136.599,170.065,50.010,159.670
C06139=1019.810,294.654,-136.631,170.070,50.007,159.670
C06140=1019.816,294.902,-136.663,170.075,50.003,159.670
C06141=1019.822,295.150,-136.694,170.080,50.000,159.670
C06142=1019.828,295.398,-136.726,170.086,49.996,159.670
C06143=1019.834,295.645,-136.758,170.091,49.992,159.670
C06144=1019.841,295.893,-136.790,170.096,49.988,159.670
C06145=1019.847,296.142,-136.822,170.102,49.985,159.670
C06146=1019.854,296.389,-136.853,170.106,49.981,159.670
C06147=1019.860,296.638,-136.885,170.112,49.978,159.670
C06148=1019.866,296.884,-136.917,170.118,49.974,159.670
C06149=1019.872,297.132,-136.949,170.123,49.970,159.670
C06150=1019.878,297.381,-136.981,170.128,49.967,159.670
C06151=1019.885,297.628,-137.013,170.133,49.963,159.670
C06152=1019.891,297.876,-137.045,170.138,49.960,159.670
C06153=1019.898,298.124,-137.077,170.144,49.956,159.670
C06154=1019.904,298.372,-137.110,170.150,49.952,159.670
C06155=1019.911,298.620,-137.141,170.155,49.949,159.670
C06156=1019.917,298.868,-137.173,170.160,49.946,159.670
C06157=1019.923,299.115,-137.206,170.165,49.942,159.671
C06158=1019.930,299.363,-137.237,170.170,49.938,159.670
C06159=1019.936,299.611,-137.269,170.177,49.935,159.671
C06160=1019.943,299.859,-137.301,170.182,49.931,159.671
C06161=1019.949,300.107,-137.333,170.187,49.928,159.671
C06162=1019.956,300.354,-137.366,170.192,49.924,159.671
C06163=1019.962,300.602,-137.398,170.197,49.921,159.671
C06164=1019.968,300.850,-137.430,170.204,49.917,159.671
C06165=1019.975,301.098,-137.462,170.209,49.914,159.671
C06166=1019.981,301.346,-137.495,170.214,49.911,159.671
C06167=1019.988,301.593,-137.526,170.219,49.907,159.671
C06168=1019.994,301.841,-137.559,170.225,49.903,159.671
C06169=1020.001,302.089,-137.591,170.231,49.900,159.671
C06170=1020.007,302.337,-137.623,170.236,49.896,159.672
C06171=1020.014,302.585,-137.656,170.241,49.893,159.672
C06172=1020.021,302.833,-137.687,170.247,49.890,159.672
C06173=1020.027,303.080,-137.720,170.252,49.887,159.672
C06174=1020.034,303.328,-137.752,170.258,49.883,159.672
C06175=1020.040,303.576,-137.784,170.264,49.880,159.672
C06176=1020.047,303.823,-137.817,170.268,49.876,159.672
C06177=1020.054,304.071,-137.849,170.274,49.872,159.672
C06178=1020.060,304.320,-137.882,170.280,49.869,159.672
C06179=1020.067,304.567,-137.914,170.285,49.866,159.672
C06180=1020.073,304.814,-137.946,170.291,49.862,159.673
C06181=1020.080,305.062,-137.979,170.296,49.859,159.673
C06182=1020.087,305.309,-138.011,170.302,49.855,159.673
C06183=1020.093,305.558,-138.044,170.308,49.853,159.673
C06184=1020.100,305.806,-138.076,170.313,49.849,159.673
C06185=1020.107,306.053,-138.109,170.318,49.846,159.673
C06186=1020.113,306.301,-138.141,170.325,49.843,159.674
C06187=1020.121,306.549,-138.174,170.330,49.839,159.674
C06188=1020.127,306.796,-138.207,170.335,49.836,159.674
C06189=1020.133,307.038,-138.238,170.341,49.833,159.674
C06190=1020.140,307.279,-138.270,170.346,49.829,159.674
C06191=1020.147,307.521,-138.301,170.353,49.826,159.674
C06192=1020.154,307.761,-138.333,170.358,49.823,159.674
C06193=1020.160,308.003,-138.365,170.363,49.820,159.675
C06194=1020.166,308.245,-138.396,170.368,49.817,159.675
C06195=1020.173,308.485,-138.428,170.374,49.813,159.675
C06196=1020.180,308.727,-138.460,170.379,49.811,159.675
C06197=1020.186,308.975,-138.493,170.385,49.807,159.675
C06198=1020.193,309.223,-138.526,170.391,49.804,159.675
C06199=1020.200,309.470,-138.558,170.396,49.800,159.675
C06200=1020.207,309.718,-138.591,170.402,49.798,159.676
C06201=1020.214,309.966,-138.623,170.408,49.794,159.676
C06202=1020.220,310.213,-138.657,170.414,49.792,159.676
C06203=1020.226,310.461,-138.690,170.419,49.788,159.676
C06204=1020.234,310.708,-138.724,170.425,49.786,159.677
C06205=1020.240,310.956,-138.757,170.430,49.782,159.677
C06206=1020.247,311.203,-138.790,170.437,49.779,159.677
C06207=1020.253,311.452,-138.824,170.442,49.776,159.677
C06208=1020.259,311.699,-138.856,170.448,49.774,159.677
C06209=1020.266,311.946,-138.890,170.453,49.771,159.678
C06210=1020.272,312.194,-138.923,170.459,49.768,159.678
C06211=1020.278,312.442,-138.957,170.465,49.765,159.678
C06212=1020.286,312.689,-138.991,170.471,49.761,159.678
C06213=1020.292,312.937,-139.024,170.476,49.759,159.679
C06214=1020.299,313.185,-139.057,170.482,49.756,159.679
C06215=1020.305,313.433,-139.091,170.488,49.753,159.679
C06216=1020.312,313.680,-139.125,170.494,49.750,159.679
C06217=1020.318,313.928,-139.157,170.500,49.747,159.680
C06218=1020.325,314.176,-139.191,170.505,49.745,159.680
C06219=1020.331,314.423,-139.225,170.511,49.741,159.680
C06220=1020.338,314.671,-139.258,170.517,49.738,159.681
C06221=1020.345,314.918,-139.292,170.523,49.736,159.681
C06222=1020.352,315.166,-139.326,170.529,49.733,159.681
C06223=1020.358,315.413,-139.360,170.534,49.731,159.681
C06224=1020.365,315.661,-139.393,170.541,49.727,159.682
C06225=1020.371,315.908,-139.426,170.546,49.724,159.682
C06226=1020.378,316.156,-139.460,170.552,49.722,159.682
C06227=1020.385,316.404,-139.495,170.558,49.719,159.682
C06228=1020.391,316.652,-139.527,170.564,49.716,159.683
C06229=1020.398,316.899,-139.561,170.570,49.713,159.683
C06230=1020.405,317.146,-139.595,170.575,49.711,159.683
C06231=1020.411,317.394,-139.629,170.581,49.708,159.684
C06232=1020.419,317.642,-139.663,170.587,49.705,159.684
C06233=1020.425,317.889,-139.696,170.593,49.702,159.684
C06234=1020.432,318.136,-139.730,170.599,49.699,159.684
C06235=1020.439,318.384,-139.765,170.605,49.696,159.685
C06236=1020.446,318.633,-139.798,170.611,49.694,159.685
C06237=1020.452,318.880,-139.831,170.617,49.691,159.685
C06238=1020.460,319.127,-139.865,170.622,49.688,159.686
C06239=1020.466,319.375,-139.899,170.629,49.686,159.686
C06240=1020.473,319.622,-139.933,170.635,49.683,159.686
C06241=1020.480,319.870,-139.967,170.641,49.681,159.687
C06242=1020.487,320.118,-140.000,170.647,49.678,159.687
C06243=1020.493,320.366,-140.035,170.653,49.675,159.688
C06244=1020.501,320.613,-140.069,170.659,49.673,159.688
C06245=1020.508,320.860,-140.103,170.665,49.670,159.688
C06246=1020.514,321.108,-140.137,170.671,49.667,159.689
C06247=1020.521,321.355,-140.171,170.677,49.665,159.689
C06248=1020.528,321.603,-140.205,170.683,49.662,159.689
C06249=1020.535,321.847,-140.238,170.689,49.660,159.690
C06250=1020.542,322.091,-140.272,170.695,49.657,159.690
C06251=1020.549,322.335,-140.306,170.701,49.654,159.690
C06252=1020.555,322.579,-140.339,170.707,49.651,159.691
C06253=1020.563,322.822,-140.373,170.713,49.649,159.691
C06254=1020.569,323.066,-140.407,170.719,49.647,159.691
C06255=1020.577,323.310,-140.440,170.725,49.644,159.692
C06256=1020.584,323.554,-140.474,170.731,49.641,159.692
C06257=1020.590,323.802,-140.508,170.737,49.639,159.693
C06258=1020.598,324.049,-140.542,170.744,49.636,159.693
C06259=1020.605,324.297,-140.576,170.750,49.634,159.693
C06260=1020.612,324.544,-140.610,170.756,49.632,159.694
C06261=1020.619,324.792,-140.645,170.762,49.629,159.694
C06262=1020.626,325.039,-140.679,170.768,49.626,159.694
C06263=1020.633,325.286,-140.714,170.774,49.624,159.695
C06264=1020.640,325.535,-140.748,170.781,49.621,159.695
C06265=1020.648,325.783,-140.782,170.787,49.619,159.696
C06266=1020.655,326.030,-140.817,170.794,49.616,159.696
C06267=1020.662,326.278,-140.851,170.799,49.614,159.696
C06268=1020.669,326.525,-140.886,170.805,49.612,159.697
C06269=1020.677,326.772,-140.920,170.812,49.609,159.697
C06270=1020.683,327.020,-140.955,170.818,49.607,159.698
C06271=1020.690,327.267,-140.990,170.825,49.604,159.698
C06272=1020.697,327.515,-141.025,170.831,49.602,159.699
C06273=1020.704,327.762,-141.060,170.837,49.600,159.699
C06274=1020.711,328.010,-141.094,170.844,49.597,159.700
C06275=1020.717,328.257,-141.129,170.849,49.595,159.700
C06276=1020.725,328.504,-141.164,170.855,49.593,159.700
C06277=1020.732,328.752,-141.199,170.862,49.591,159.701
C06278=1020.739,328.999,-141.234,170.868,49.589,159.702
C06279=1020.746,329.247,-141.269,170.874,49.586,159.702
C06280=1020.753,329.494,-141.304,170.881,49.584,159.702
C06281=1020.760,329.742,-141.338,170.887,49.582,159.703
C06282=1020.767,329.989,-141.373,170.894,49.579,159.703
C06283=1020.774,330.237,-141.409,170.900,49.577,159.704
C06284=1020.781,330.484,-141.444,170.906,49.575,159.704
C06285=1020.788,330.732,-141.479,170.913,49.572,159.705
C06286=1020.795,330.979,-141.514,170.919,49.570,159.705
C06287=1020.802,331.226,-141.549,170.926,49.568,159.706
C06288=1020.810,331.474,-141.585,170.932,49.566,159.706
C06289=1020.817,331.721,-141.620,170.939,49.564,159.707
C06290=1020.824,331.968,-141.655,170.945,49.562,159.707
C06291=1020.831,332.216,-141.690,170.951,49.560,159.708
C06292=1020.839,332.463,-141.725,170.958,49.558,159.708
C06293=1020.845,332.711,-141.760,170.964,49.556,159.709
C06294=1020.853,332.959,-141.795,170.971,49.553,159.709
C06295=1020.860,333.206,-141.831,170.977,49.551,159.710
C06296=1020.867,333.453,-141.866,170.984,49.549,159.711
C06297=1020.874,333.701,-141.902,170.990,49.547,159.711
C06298=1020.881,333.948,-141.938,170.997,49.546,159.712
C06299=1020.888,334.195,-141.973,171.004,49.543,159.712
C06300=1020.895,334.443,-142.008,171.010,49.541,159.713
C06301=1020.902,334.690,-142.044,171.017,49.539,159.713
C06302=1020.909,334.937,-142.079,171.023,49.537,159.714
C06303=1020.917,335.185,-142.116,171.030,49.535,159.715
C06304=1020.923,335.432,-142.151,171.036,49.533,159.715
C06305=1020.931,335.680,-142.187,171.043,49.531,159.716
C06306=1020.938,335.927,-142.222,171.049,49.529,159.716
C06307=1020.945,336.174,-142.258,171.056,49.528,159.717
C06308=1020.952,336.422,-142.293,171.063,49.526,159.717
C06309=1020.959,336.663,-142.329,171.069,49.524,159.718
C06310=1020.967,336.905,-142.363,171.076,49.522,159.719
C06311=1020.974,337.146,-142.398,171.082,49.520,159.719
C06312=1020.981,337.388,-142.433,171.088,49.518,159.720
C06313=1020.988,337.630,-142.468,171.095,49.516,159.720
C06314=1020.995,337.872,-142.504,171.101,49.514,159.721
C06315=1021.002,338.114,-142.538,171.108,49.513,159.721
C06316=1021.009,338.355,-142.574,171.115,49.511,159.722
C06317=1021.016,338.602,-142.610,171.121,49.509,159.723
C06318=1021.024,338.850,-142.645,171.128,49.507,159.723
C06319=1021.031,339.097,-142.681,171.135,49.506,159.724
C06320=1021.039,339.344,-142.717,171.142,49.503,159.725
C06321=1021.046,339.591,-142.753,171.148,49.502,159.725
C06322=1021.053,339.838,-142.789,171.155,49.500,159.726
C06323=1021.061,340.086,-142.826,171.161,49.498,159.726
C06324=1021.068,340.333,-142.862,171.169,49.497,159.727
C06325=1021.075,340.580,-142.898,171.175,49.495,159.728
C06326=1021.083,340.828,-142.934,171.182,49.493,159.728
C06327=1021.090,341.075,-142.971,171.189,49.492,159.729
C06328=1021.097,341.322,-143.007,171.196,49.489,159.730
C06329=1021.104,341.570,-143.043,171.202,49.488,159.730
C06330=1021.112,341.817,-143.080,171.209,49.486,159.731
C06331=1021.119,342.064,-143.115,171.217,49.485,159.732
C06332=1021.126,342.312,-143.152,171.223,49.483,159.733
C06333=1021.134,342.558,-143.189,171.230,49.481,159.733
C06334=1021.142,342.806,-143.225,171.237,49.480,159.734
C06335=1021.149,343.053,-143.261,171.244,49.478,159.735
C06336=1021.156,343.300,-143.298,171.250,49.477,159.735
C06337=1021.164,343.547,-143.335,171.258,49.475,159.736
C06338=1021.171,343.795,-143.372,171.265,49.473,159.737
C06339=1021.178,344.042,-143.408,171.272,49.472,159.738
C06340=1021.186,344.288,-143.445,171.279,49.470,159.738
C06341=1021.193,344.536,-143.481,171.285,49.469,159.739
C06342=1021.200,344.784,-143.518,171.293,49.467,159.740
C06343=1021.208,345.030,-143.554,171.299,49.466,159.740
C06344=1021.215,345.278,-143.591,171.307,49.464,159.741
C06345=1021.223,345.525,-143.628,171.314,49.462,159.742
C06346=1021.231,345.772,-143.664,171.320,49.461,159.743
C06347=1021.238,346.020,-143.702,171.328,49.459,159.743
C06348=1021.246,346.267,-143.738,171.335,49.458,159.744
C06349=1021.254,346.514,-143.775,171.341,49.456,159.745
C06350=1021.261,346.762,-143.812,171.349,49.455,159.746
C06351=1021.268,347.008,-143.848,171.357,49.454,159.747
C06352=1021.275,347.255,-143.886,171.363,49.452,159.747
C06353=1021.283,347.502,-143.922,171.370,49.451,159.748
C06354=1021.290,347.749,-143.960,171.377,49.449,159.749
C06355=1021.298,347.996,-143.997,171.385,49.448,159.750
C06356=1021.305,348.244,-144.033,171.392,49.446,159.750
C06357=1021.313,348.491,-144.070,171.398,49.445,159.751
C06358=1021.320,348.738,-144.108,171.406,49.444,159.752
C06359=1021.329,348.986,-144.145,171.413,49.442,159.753
C06360=1021.336,349.233,-144.183,171.420,49.441,159.753
C06361=1021.343,349.480,-144.220,171.428,49.440,159.754
C06362=1021.351,349.727,-144.257,171.435,49.438,159.755
C06363=1021.359,349.974,-144.295,171.442,49.438,159.756
C06364=1021.367,350.221,-144.332,171.449,49.436,159.757
C06365=1021.374,350.468,-144.369,171.457,49.435,159.758
C06366=1021.381,350.715,-144.407,171.464,49.433,159.758
C06367=1021.389,350.962,-144.444,171.471,49.432,159.759
C06368=1021.396,351.209,-144.481,171.478,49.431,159.760
C06369=1021.404,351.449,-144.518,171.485,49.430,159.761
C06370=1021.411,351.690,-144.554,171.493,49.428,159.762
C06371=1021.419,351.930,-144.591,171.500,49.427,159.763
C06372=1021.427,352.170,-144.628,171.507,49.426,159.764
C06373=1021.434,352.410,-144.663,171.514,49.425,159.764
C06374=1021.441,352.650,-144.700,171.521,49.424,159.765
C06375=1021.449,352.890,-144.737,171.529,49.422,159.766
C06376=1021.457,353.130,-144.774,171.535,49.422,159.767
C06377=1021.465,353.377,-144.811,171.543,49.421,159.768
C06378=1021.472,353.624,-144.848,171.551,49.420,159.769
C06379=1021.480,353.872,-144.886,171.558,49.418,159.770
C06380=1021.488,354.118,-144.924,171.566,49.417,159.771
C06381=1021.495,354.365,-144.961,171.573,49.416,159.771
C06382=1021.503,354.613,-145.000,171.580,49.415,159.772
C06383=1021.511,354.860,-145.037,171.588,49.414,159.773
C06384=1021.518,355.106,-145.075,171.596,49.413,159.774
C06385=1021.527,355.354,-145.113,171.603,49.412,159.775
C06386=1021.534,355.600,-145.151,171.610,49.411,159.776
C06387=1021.542,355.847,-145.189,171.618,49.410,159.777
C06388=1021.550,356.095,-145.227,171.626,49.409,159.778
C06389=1021.557,356.341,-145.265,171.634,49.408,159.779
C06390=1021.566,356.589,-145.303,171.641,49.407,159.780
C06391=1021.573,356.835,-145.341,171.648,49.406,159.781
C06392=1021.582,357.082,-145.380,171.656,49.405,159.782
C06393=1021.589,357.329,-145.418,171.664,49.404,159.783
C06394=1021.597,357.577,-145.456,171.671,49.403,159.784
C06395=1021.605,357.823,-145.494,171.679,49.402,159.785
C06396=1021.613,358.071,-145.533,171.687,49.401,159.786
C06397=1021.621,358.317,-145.570,171.695,49.400,159.787
C06398=1021.629,358.564,-145.609,171.702,49.399,159.788
C06399=1021.637,358.811,-145.647,171.710,49.398,159.789
C06400=1021.645,359.058,-145.686,171.717,49.397,159.790
C06401=1021.652,359.304,-145.724,171.725,49.397,159.791
C06402=1021.661,359.551,-145.763,171.733,49.396,159.792
C06403=1021.669,359.799,-145.801,171.741,49.395,159.793
C06404=1021.676,360.045,-145.839,171.749,49.394,159.794
C06405=1021.684,360.292,-145.878,171.757,49.393,159.795
C06406=1021.692,360.539,-145.916,171.764,49.392,159.796
C06407=1021.700,360.786,-145.955,171.773,49.392,159.797
C06408=1021.708,361.034,-145.994,171.780,49.391,159.798
C06409=1021.715,361.280,-146.033,171.787,49.390,159.799
C06410=1021.724,361.527,-146.072,171.795,49.389,159.800
C06411=1021.732,361.774,-146.110,171.803,49.389,159.801
C06412=1021.740,362.020,-146.149,171.811,49.388,159.802
C06413=1021.748,362.267,-146.188,171.819,49.387,159.803
C06414=1021.756,362.514,-146.226,171.827,49.387,159.804
C06415=1021.764,362.761,-146.266,171.835,49.386,159.805
C06416=1021.771,363.008,-146.305,171.843,49.385,159.806
C06417=1021.780,363.254,-146.344,171.851,49.385,159.808
C06418=1021.788,363.502,-146.382,171.859,49.384,159.809
C06419=1021.796,363.748,-146.422,171.867,49.383,159.810
C06420=1021.804,363.995,-146.460,171.875,49.383,159.811
C06421=1021.811,364.242,-146.500,171.883,49.382,159.812
C06422=1021.820,364.489,-146.539,171.891,49.382,159.813
C06423=1021.828,364.735,-146.578,171.899,49.381,159.814
C06424=1021.837,364.982,-146.617,171.907,49.380,159.815
C06425=1021.845,365.229,-146.656,171.915,49.380,159.816
C06426=1021.853,365.476,-146.695,171.924,49.379,159.818
C06427=1021.861,365.723,-146.735,171.933,49.379,159.819
C06428=1021.869,365.969,-146.774,171.941,49.378,159.820
C06429=1021.877,366.213,-146.813,171.949,49.378,159.821
C06430=1021.885,366.457,-146.851,171.957,49.377,159.822
C06431=1021.893,366.700,-146.890,171.965,49.377,159.823
C06432=1021.902,366.944,-146.929,171.973,49.376,159.825
C06433=1021.910,367.187,-146.968,171.981,49.376,159.826
C06434=1021.919,367.431,-147.006,171.989,49.375,159.827
C06435=1021.927,367.675,-147.046,171.997,49.375,159.828
C06436=1021.935,367.918,-147.084,172.006,49.374,159.829
C06437=1021.943,368.165,-147.124,172.014,49.374,159.830
C06438=1021.951,368.412,-147.163,172.022,49.373,159.832
C06439=1021.959,368.658,-147.203,172.030,49.374,159.833
C06440=1021.968,368.904,-147.243,172.038,49.373,159.834
C06441=1021.976,369.152,-147.284,172.048,49.372,159.835
C06442=1021.984,369.399,-147.323,172.056,49.372,159.836
C06443=1021.992,369.646,-147.363,172.064,49.372,159.838
C06444=1022.001,369.891,-147.403,172.072,49.372,159.839
C06445=1022.009,370.138,-147.443,172.081,49.372,159.840
C06446=1022.017,370.385,-147.482,172.089,49.371,159.841
C06447=1022.025,370.631,-147.523,172.098,49.371,159.843
C06448=1022.034,370.879,-147.562,172.106,49.370,159.844
C06449=1022.042,371.125,-147.603,172.115,49.371,159.845
C06450=1022.051,371.371,-147.642,172.123,49.370,159.847
C06451=1022.059,371.618,-147.683,172.132,49.370,159.848
C06452=1022.068,371.865,-147.723,172.141,49.369,159.849
C06453=1022.076,372.111,-147.763,172.149,49.370,159.851
C06454=1022.084,372.358,-147.803,172.157,49.369,159.852
C06455=1022.092,372.604,-147.843,172.167,49.369,159.853
C06456=1022.102,372.851,-147.884,172.175,49.369,159.854
C06457=1022.109,373.098,-147.924,172.183,49.368,159.856
C06458=1022.118,373.344,-147.964,172.192,49.369,159.857
C06459=1022.127,373.591,-148.005,172.201,49.368,159.858
C06460=1022.135,373.837,-148.044,172.210,49.369,159.860
C06461=1022.144,374.084,-148.085,172.218,49.368,159.861
C06462=1022.153,374.330,-148.125,172.227,49.368,159.862
C06463=1022.161,374.577,-148.166,172.236,49.368,159.864
C06464=1022.170,374.823,-148.206,172.245,49.368,159.865
C06465=1022.178,375.071,-148.246,172.254,49.368,159.867
C06466=1022.187,375.317,-148.286,172.262,49.368,159.868
C06467=1022.196,375.564,-148.327,172.272,49.368,159.869
C06468=1022.204,375.810,-148.368,172.280,49.368,159.871
C06469=1022.213,376.057,-148.409,172.288,49.368,159.872
C06470=1022.222,376.303,-148.449,172.298,49.368,159.873
C06471=1022.230,376.550,-148.490,172.306,49.368,159.875
C06472=1022.239,376.795,-148.531,172.316,49.368,159.876
C06473=1022.247,377.042,-148.572,172.324,49.368,159.878
C06474=1022.256,377.288,-148.612,172.334,49.368,159.879
C06475=1022.265,377.535,-148.654,172.342,49.368,159.880
C06476=1022.274,377.782,-148.695,172.351,49.368,159.882
C06477=1022.282,378.028,-148.735,172.361,49.368,159.883
C06478=1022.291,378.274,-148.777,172.369,49.368,159.885
C06479=1022.299,378.521,-148.818,172.379,49.369,159.886
C06480=1022.308,378.767,-148.859,172.387,49.369,159.888
C06481=1022.317,379.014,-148.900,172.397,49.368,159.889
C06482=1022.326,379.260,-148.941,172.406,49.369,159.891
C06483=1022.334,379.506,-148.982,172.415,49.369,159.892
C06484=1022.343,379.753,-149.024,172.424,49.370,159.894
C06485=1022.352,380.000,-149.065,172.433,49.369,159.895
C06486=1022.361,380.246,-149.107,172.442,49.370,159.897
C06487=1022.370,380.491,-149.147,172.452,49.370,159.898
C06488=1022.378,380.738,-149.188,172.461,49.371,159.900
C06489=1022.387,380.982,-149.229,172.470,49.370,159.901
C06490=1022.396,381.226,-149.271,172.479,49.371,159.903
C06491=1022.404,381.470,-149.311,172.488,49.371,159.904
C06492=1022.413,381.713,-149.353,172.498,49.371,159.906
C06493=1022.423,381.957,-149.394,172.507,49.372,159.907
C06494=1022.431,382.201,-149.435,172.517,49.372,159.909
C06495=1022.440,382.445,-149.476,172.525,49.372,159.910
C06496=1022.449,382.689,-149.517,172.535,49.373,159.912
C06497=1022.458,382.935,-149.559,172.544,49.373,159.914
C06498=1022.467,383.181,-149.600,172.554,49.373,159.915
C06499=1022.476,383.428,-149.642,172.563,49.373,159.917
C06500=1022.485,383.674,-149.683,172.573,49.374,159.918
C06501=1022.494,383.920,-149.725,172.582,49.374,159.920
C06502=1022.504,384.166,-149.767,172.592,49.375,159.922
C06503=1022.512,384.412,-149.809,172.602,49.375,159.923
C06504=1022.521,384.659,-149.851,172.611,49.376,159.925
C06505=1022.530,384.905,-149.892,172.620,49.376,159.926
C06506=1022.540,385.151,-149.934,172.630,49.377,159.928
C06507=1022.549,385.397,-149.976,172.640,49.377,159.930
C06508=1022.559,385.644,-150.018,172.650,49.377,159.931
C06509=1022.568,385.890,-150.060,172.659,49.378,159.933
C06510=1022.577,386.136,-150.102,172.669,49.379,159.935
C06511=1022.586,386.382,-150.144,172.679,49.379,159.936
C06512=1022.594,386.628,-150.187,172.689,49.380,159.938
C06513=1022.604,386.876,-150.229,172.698,49.380,159.940
C06514=1022.613,387.121,-150.272,172.708,49.381,159.942
C06515=1022.622,387.367,-150.314,172.718,49.381,159.943
C06516=1022.631,387.613,-150.356,172.727,49.382,159.945
C06517=1022.641,387.860,-150.398,172.738,49.383,159.947
C06518=1022.650,388.106,-150.441,172.747,49.383,159.948
C06519=1022.659,388.352,-150.483,172.758,49.384,159.950
C06520=1022.668,388.599,-150.526,172.767,49.384,159.952
C06521=1022.678,388.844,-150.568,172.778,49.385,159.954
C06522=1022.687,389.090,-150.611,172.788,49.386,159.956
C06523=1022.697,389.337,-150.654,172.797,49.387,159.957
C06524=1022.706,389.582,-150.696,172.807,49.388,159.959
C06525=1022.715,389.828,-150.739,172.817,49.389,159.961
C06526=1022.724,390.075,-150.782,172.827,49.389,159.962
C06527=1022.734,390.321,-150.824,172.837,49.390,159.964
C06528=1022.743,390.567,-150.868,172.847,49.391,159.966
C06529=1022.752,390.813,-150.910,172.858,49.392,159.968
C06530=1022.762,391.059,-150.954,172.867,49.392,159.970
C06531=1022.771,391.305,-150.996,172.878,49.393,159.971
C06532=1022.780,391.551,-151.040,172.888,49.394,159.973
C06533=1022.791,391.818,-151.086,172.899,49.395,159.975
C06534=1022.801,392.086,-151.133,172.911,49.396,159.977
C06535=1022.812,392.353,-151.180,172.922,49.397,159.980
C06536=1022.823,392.621,-151.227,172.932,49.398,159.981
C06537=1022.832,392.866,-151.269,172.944,49.398,159.983
C06538=1022.841,393.113,-151.313,172.954,49.399,159.985
C06539=1022.851,393.359,-151.356,172.964,49.401,159.987
C06540=1022.860,393.605,-151.400,172.975,49.402,159.989
C06541=1022.870,393.851,-151.443,172.985,49.402,159.991
C06542=1022.879,394.097,-151.487,172.995,49.403,159.993
C06543=1022.889,394.342,-151.530,173.006,49.405,159.995
C06544=1022.898,394.589,-151.573,173.017,49.405,159.997
C06545=1022.908,394.835,-151.617,173.027,49.406,159.999
C06546=1022.918,395.081,-151.660,173.038,49.408,160.001
C06547=1022.927,395.326,-151.704,173.048,49.409,160.003
C06548=1022.937,395.572,-151.748,173.059,49.410,160.005
C06549=1022.949,395.872,-151.801,173.072,49.411,160.007
C06550=1022.961,396.172,-151.854,173.085,49.413,160.010
C06551=1022.972,396.471,-151.907,173.098,49.414,160.012
C06552=1022.984,396.770,-151.961,173.111,49.415,160.014
C06553=1022.994,397.016,-152.005,173.121,49.416,160.016
C06554=1023.004,397.262,-152.048,173.133,49.417,160.018
C06555=1023.013,397.507,-152.093,173.143,49.419,160.020
C06556=1023.024,397.753,-152.136,173.154,49.420,160.022
C06557=1023.033,397.999,-152.181,173.165,49.421,160.024
C06558=1023.043,398.245,-152.224,173.176,49.422,160.026
C06559=1023.053,398.491,-152.269,173.186,49.424,160.029
C06560=1023.063,398.736,-152.312,173.198,49.425,160.031
C06561=1023.073,398.983,-152.358,173.209,49.426,160.033
C06562=1023.083,399.229,-152.402,173.220,49.427,160.035
C06563=1023.093,399.474,-152.446,173.231,49.429,160.037
C06564=1023.103,399.720,-152.490,173.242,49.430,160.039
C06565=1023.112,399.966,-152.535,173.253,49.431,160.041
C06566=1023.122,400.212,-152.578,173.264,49.433,160.043
C06567=1023.132,400.457,-152.623,173.275,49.434,160.045
C06568=1023.142,400.703,-152.668,173.287,49.435,160.048
C06569=1023.153,400.948,-152.713,173.298,49.437,160.050
C06570=1023.162,401.195,-152.757,173.309,49.438,160.052
C06571=1023.172,401.440,-152.802,173.320,49.440,160.054
C06572=1023.182,401.686,-152.847,173.332,49.441,160.056
C06573=1023.192,401.932,-152.892,173.343,49.442,160.058
C06574=1023.202,402.177,-152.936,173.354,49.444,160.061
C06575=1023.213,402.423,-152.981,173.366,49.446,160.063
C06576=1023.223,402.669,-153.026,173.377,49.448,160.065
C06577=1023.233,402.914,-153.071,173.388,49.449,160.067
C06578=1023.243,403.160,-153.117,173.400,49.450,160.070
C06579=1023.253,403.405,-153.161,173.411,49.452,160.072
C06580=1023.263,403.652,-153.207,173.423,49.453,160.074
C06581=1023.273,403.897,-153.251,173.435,49.455,160.076
C06582=1023.283,404.143,-153.297,173.447,49.457,160.079
C06583=1023.294,404.388,-153.342,173.457,49.458,160.081
C06584=1023.304,404.634,-153.387,173.469,49.460,160.083
C06585=1023.314,404.879,-153.432,173.481,49.461,160.086
C06586=1023.324,405.125,-153.477,173.493,49.463,160.088
C06587=1023.335,405.371,-153.523,173.504,49.465,160.090
C06588=1023.345,405.616,-153.568,173.516,49.467,160.093
C06589=1023.355,405.862,-153.614,173.528,49.468,160.095
C06590=1023.367,406.107,-153.659,173.540,49.470,160.097
C06591=1023.376,406.353,-153.704,173.552,49.472,160.100
C06592=1023.387,406.598,-153.750,173.564,49.473,160.102
C06593=1023.398,406.844,-153.796,173.576,49.475,160.104
C06594=1023.408,407.090,-153.841,173.588,49.477,160.107
C06595=1023.419,407.336,-153.887,173.600,49.478,160.109
C06596=1023.429,407.581,-153.933,173.612,49.480,160.112
C06597=1023.439,407.826,-153.979,173.624,49.482,160.114
C06598=1023.451,408.071,-154.024,173.636,49.484,160.116
C06599=1023.461,408.317,-154.070,173.648,49.486,160.119
C06600=1023.472,408.563,-154.116,173.660,49.487,160.121
C06601=1023.482,408.808,-154.162,173.672,49.489,160.124
C06602=1023.493,409.054,-154.208,173.684,49.491,160.126
C06603=1023.504,409.299,-154.253,173.696,49.493,160.129
C06604=1023.514,409.545,-154.299,173.709,49.495,160.131
C06605=1023.525,409.791,-154.345,173.721,49.497,160.134
C06606=1023.536,410.036,-154.392,173.733,49.499,160.136
C06607=1023.546,410.282,-154.439,173.745,49.501,160.139
C06608=1023.557,410.528,-154.485,173.759,49.503,160.141
C06609=1023.572,410.850,-154.545,173.775,49.506,160.145
C06610=1023.585,411.172,-154.607,173.791,49.508,160.148
C06611=1023.600,411.493,-154.667,173.808,49.511,160.151
C06612=1023.614,411.816,-154.729,173.824,49.514,160.155
C06613=1023.625,412.061,-154.775,173.836,49.516,160.157
C06614=1023.635,412.306,-154.821,173.850,49.518,160.160
C06615=1023.646,412.552,-154.869,173.862,49.520,160.163
C06616=1023.657,412.797,-154.916,173.874,49.522,160.165
C06617=1023.668,413.042,-154.962,173.888,49.524,160.168
C06618=1023.679,413.288,-155.009,173.900,49.527,160.171
C06619=1023.690,413.533,-155.056,173.913,49.529,160.173
C06620=1023.700,413.778,-155.103,173.926,49.531,160.176
C06621=1023.712,414.024,-155.150,173.939,49.533,160.179
C06622=1023.723,414.269,-155.197,173.952,49.535,160.181
C06623=1023.734,414.514,-155.244,173.964,49.537,160.184
C06624=1023.745,414.759,-155.290,173.978,49.540,160.187
C06625=1023.756,415.005,-155.338,173.991,49.542,160.189
C06626=1023.768,415.251,-155.385,174.004,49.544,160.192
C06627=1023.779,415.496,-155.431,174.017,49.547,160.195
C06628=1023.790,415.741,-155.480,174.030,49.549,160.198
C06629=1023.801,415.987,-155.527,174.044,49.551,160.200
C06630=1023.812,416.231,-155.574,174.057,49.554,160.203
C06631=1023.823,416.477,-155.622,174.070,49.556,160.206
C06632=1023.835,416.722,-155.669,174.084,49.558,160.209
C06633=1023.846,416.967,-155.717,174.097,49.561,160.212
C06634=1023.857,417.213,-155.764,174.110,49.563,160.215
C06635=1023.868,417.458,-155.812,174.124,49.566,160.217
C06636=1023.879,417.702,-155.860,174.137,49.568,160.220
C06637=1023.891,417.948,-155.908,174.151,49.571,160.223
C06638=1023.902,418.193,-155.955,174.164,49.573,160.226
C06639=1023.913,418.439,-156.003,174.178,49.575,160.229
C06640=1023.925,418.684,-156.051,174.192,49.578,160.232
C06641=1023.936,418.929,-156.099,174.205,49.581,160.235
C06642=1023.948,419.174,-156.147,174.218,49.583,160.238
C06643=1023.959,419.420,-156.195,174.233,49.586,160.241
C06644=1023.971,419.664,-156.244,174.246,49.588,160.244
C06645=1023.983,419.909,-156.292,174.260,49.591,160.247
C06646=1023.994,420.155,-156.340,174.274,49.593,160.249
C06647=1024.006,420.400,-156.388,174.288,49.596,160.253
C06648=1024.017,420.644,-156.437,174.302,49.599,160.255
C06649=1024.029,420.889,-156.484,174.316,49.601,160.259
C06650=1024.040,421.135,-156.533,174.330,49.604,160.262
C06651=1024.052,421.379,-156.581,174.344,49.607,160.265
C06652=1024.064,421.625,-156.630,174.358,49.609,160.268
C06653=1024.076,421.870,-156.678,174.372,49.612,160.271
C06654=1024.087,422.115,-156.726,174.387,49.615,160.274
C06655=1024.099,422.360,-156.775,174.401,49.618,160.277
C06656=1024.111,422.604,-156.824,174.415,49.620,160.280
C06657=1024.123,422.850,-156.873,174.429,49.623,160.283
C06658=1024.134,423.094,-156.922,174.444,49.627,160.286
C06659=1024.147,423.339,-156.971,174.459,49.629,160.290
C06660=1024.159,423.584,-157.020,174.473,49.632,160.293
C06661=1024.170,423.829,-157.069,174.487,49.635,160.296
C06662=1024.183,424.074,-157.118,174.503,49.638,160.299
C06663=1024.194,424.319,-157.167,174.517,49.640,160.302
C06664=1024.206,424.564,-157.216,174.531,49.643,160.305
C06665=1024.218,424.809,-157.265,174.546,49.646,160.309
C06666=1024.230,425.054,-157.314,174.561,49.650,160.312
C06667=1024.242,425.298,-157.364,174.576,49.652,160.315
C06668=1024.255,425.543,-157.412,174.590,49.655,160.318
C06669=1024.271,425.877,-157.480,174.611,49.659,160.323
C06670=1024.287,426.211,-157.548,174.631,49.663,160.327
C06671=1024.304,426.543,-157.615,174.651,49.668,160.332
C06672=1024.320,426.876,-157.683,174.672,49.671,160.336
C06673=1024.333,427.121,-157.733,174.687,49.675,160.340
C06674=1024.345,427.366,-157.783,174.702,49.678,160.343
C06675=1024.357,427.610,-157.832,174.718,49.681,160.347
C06676=1024.369,427.856,-157.882,174.733,49.684,160.350
C06677=1024.381,428.100,-157.932,174.748,49.688,160.353
C06678=1024.393,428.345,-157.982,174.763,49.690,160.357
C06679=1024.406,428.589,-158.033,174.779,49.694,160.360
C06680=1024.418,428.834,-158.083,174.795,49.697,160.364
C06681=1024.431,429.079,-158.132,174.811,49.700,160.367
C06682=1024.444,429.324,-158.183,174.826,49.703,160.371
C06683=1024.456,429.568,-158.233,174.841,49.707,160.374
C06684=1024.468,429.813,-158.283,174.856,49.710,160.378
C06685=1024.481,430.057,-158.334,174.872,49.714,160.381
C06686=1024.493,430.302,-158.384,174.888,49.717,160.385
C06687=1024.506,430.546,-158.434,174.905,49.720,160.389
C06688=1024.518,430.791,-158.485,174.920,49.723,160.392
C06689=1024.531,431.036,-158.536,174.936,49.726,160.396
C06690=1024.544,431.280,-158.587,174.952,49.730,160.399
C06691=1024.557,431.525,-158.636,174.968,49.733,160.403
C06692=1024.570,431.769,-158.687,174.984,49.737,160.406
C06693=1024.583,432.014,-158.738,175.000,49.740,160.410
C06694=1024.595,432.258,-158.789,175.017,49.744,160.414
C06695=1024.608,432.502,-158.840,175.033,49.747,160.418
C06696=1024.621,432.747,-158.891,175.049,49.751,160.421
C06697=1024.634,432.991,-158.942,175.066,49.754,160.425
C06698=1024.647,433.236,-158.993,175.082,49.758,160.429
C06699=1024.660,433.481,-159.044,175.098,49.762,160.432
C06700=1024.673,433.725,-159.095,175.115,49.765,160.436
C06701=1024.686,433.969,-159.146,175.131,49.769,160.440
C06702=1024.699,434.214,-159.197,175.148,49.772,160.444
C06703=1024.712,434.458,-159.248,175.164,49.776,160.447
C06704=1024.724,434.703,-159.301,175.182,49.779,160.451
C06705=1024.738,434.948,-159.352,175.199,49.783,160.455
C06706=1024.751,435.191,-159.403,175.215,49.787,160.459
C06707=1024.764,435.435,-159.455,175.232,49.790,160.463
C06708=1024.777,435.680,-159.507,175.249,49.794,160.467
C06709=1024.791,435.925,-159.558,175.266,49.798,160.471
C06710=1024.803,436.169,-159.611,175.283,49.801,160.475
C06711=1024.817,436.413,-159.662,175.301,49.805,160.479
C06712=1024.830,436.657,-159.714,175.318,49.809,160.483
C06713=1024.844,436.901,-159.766,175.334,49.813,160.487
C06714=1024.857,437.146,-159.818,175.352,49.817,160.491
C06715=1024.871,437.390,-159.870,175.369,49.820,160.495
C06716=1024.883,437.635,-159.923,175.387,49.824,160.499
C06717=1024.897,437.878,-159.975,175.404,49.828,160.503
C06718=1024.911,438.122,-160.027,175.422,49.832,160.507
C06719=1024.924,438.367,-160.079,175.439,49.836,160.511
C06720=1024.937,438.611,-160.132,175.457,49.840,160.515
C06721=1024.951,438.855,-160.184,175.475,49.844,160.519
C06722=1024.965,439.099,-160.237,175.493,49.848,160.523
C06723=1024.979,439.342,-160.289,175.511,49.852,160.527
C06724=1024.992,439.588,-160.342,175.529,49.856,160.532
C06725=1025.006,439.831,-160.395,175.546,49.860,160.536
C06726=1025.020,440.075,-160.447,175.564,49.864,160.540
C06727=1025.033,440.320,-160.501,175.583,49.868,160.544
C06728=1025.047,440.563,-160.553,175.601,49.872,160.548
C06729=1025.066,440.903,-160.627,175.626,49.878,160.554
C06730=1025.086,441.242,-160.700,175.652,49.883,160.560
C06731=1025.105,441.581,-160.774,175.677,49.889,160.566
C06732=1025.125,441.920,-160.848,175.703,49.894,160.572
C06733=1025.139,442.163,-160.901,175.721,49.899,160.577
C06734=1025.153,442.406,-160.954,175.740,49.902,160.581
C06735=1025.168,442.650,-161.007,175.759,49.907,160.585
C06736=1025.182,442.894,-161.059,175.778,49.911,160.590
C06737=1025.198,443.137,-161.112,175.796,49.915,160.594
C06738=1025.214,443.380,-161.163,175.816,49.918,160.598
C06739=1025.230,443.624,-161.214,175.835,49.922,160.603
C06740=1025.247,443.868,-161.265,175.854,49.926,160.607
C06741=1025.264,444.112,-161.315,175.872,49.930,160.611
C06742=1025.282,444.355,-161.365,175.892,49.934,160.616
C06743=1025.300,444.599,-161.415,175.911,49.937,160.620
C06744=1025.319,444.843,-161.464,175.931,49.941,160.625
C06745=1025.338,445.087,-161.513,175.951,49.944,160.629
C06746=1025.357,445.332,-161.561,175.971,49.947,160.633
C06747=1025.378,445.576,-161.610,175.990,49.950,160.637
C06748=1025.398,445.820,-161.657,176.010,49.953,160.642
C06749=1025.419,446.064,-161.705,176.030,49.957,160.646
C06750=1025.439,446.309,-161.751,176.049,49.960,160.650
C06751=1025.462,446.553,-161.798,176.070,49.963,160.655
C06752=1025.483,446.798,-161.844,176.090,49.966,160.659
C06753=1025.507,447.042,-161.890,176.110,49.969,160.663
C06754=1025.529,447.287,-161.936,176.131,49.972,160.668
C06755=1025.553,447.532,-161.980,176.150,49.975,160.672
C06756=1025.577,447.777,-162.024,176.171,49.977,160.676
C06757=1025.601,448.021,-162.069,176.191,49.980,160.680
C06758=1025.626,448.267,-162.113,176.213,49.982,160.685
C06759=1025.651,448.512,-162.157,176.234,49.985,160.689
C06760=1025.677,448.757,-162.200,176.254,49.988,160.693
C06761=1025.704,449.002,-162.243,176.276,49.990,160.698
C06762=1025.730,449.248,-162.284,176.296,49.992,160.702
C06763=1025.758,449.492,-162.327,176.318,49.994,160.706
C06764=1025.785,449.738,-162.368,176.339,49.997,160.710
C06765=1025.813,449.983,-162.409,176.360,49.999,160.715
C06766=1025.841,450.228,-162.450,176.382,50.001,160.719
C06767=1025.870,450.474,-162.490,176.403,50.003,160.723
C06768=1025.900,450.719,-162.530,176.425,50.005,160.727
C06769=1025.930,450.964,-162.569,176.446,50.007,160.731
C06770=1025.959,451.210,-162.609,176.467,50.009,160.736
C06771=1025.991,451.456,-162.648,176.490,50.010,160.740
C06772=1026.022,451.701,-162.686,176.511,50.012,160.744
C06773=1025.392,448.754,-162.528,176.247,50.048,160.711
C06774=1025.367,448.510,-162.485,176.227,50.046,160.707
C06775=1025.342,448.264,-162.442,176.205,50.044,160.703
C06776=1025.317,448.019,-162.398,176.185,50.041,160.698
C06777=1025.293,447.774,-162.355,176.164,50.038,160.694
C06778=1025.268,447.530,-162.310,176.144,50.036,160.690
C06779=1025.245,447.285,-162.264,176.123,50.033,160.685
C06780=1025.222,447.040,-162.219,176.103,50.031,160.681
C06781=1025.199,446.796,-162.173,176.083,50.028,160.677
C06782=1025.177,446.550,-162.127,176.063,50.025,160.673
C06783=1025.155,446.306,-162.081,176.043,50.022,160.668
C06784=1025.134,446.061,-162.034,176.022,50.019,160.664
C06785=1025.113,445.817,-161.987,176.002,50.016,160.660
C06786=1025.092,445.573,-161.940,175.983,50.013,160.656
C06787=1025.072,445.329,-161.891,175.963,50.010,160.651
C06788=1025.052,445.085,-161.843,175.943,50.006,160.647
C06789=1025.033,444.841,-161.794,175.924,50.003,160.643
C06790=1025.015,444.596,-161.745,175.904,50.000,160.638
C06791=1024.997,444.352,-161.695,175.884,49.996,160.634
C06792=1024.980,444.108,-161.646,175.865,49.993,160.630
C06793=1024.962,443.865,-161.595,175.846,49.990,160.625
C06794=1024.944,443.621,-161.545,175.827,49.986,160.621
C06795=1024.929,443.377,-161.493,175.808,49.982,160.617
C06796=1024.913,443.134,-161.442,175.789,49.978,160.612
C06797=1024.897,442.890,-161.390,175.770,49.974,160.608
C06798=1024.881,442.646,-161.338,175.751,49.971,160.604
C06799=1024.867,442.403,-161.285,175.732,49.967,160.599
C06800=1024.853,442.160,-161.233,175.713,49.962,160.595
C06801=1024.839,441.917,-161.179,175.696,49.959,160.591
C06802=1024.821,441.607,-161.112,175.671,49.954,160.585
C06803=1024.803,441.296,-161.044,175.648,49.948,160.580
C06804=1024.785,440.985,-160.976,175.624,49.943,160.574
C06805=1024.768,440.674,-160.909,175.601,49.938,160.569
C06806=1024.754,440.430,-160.857,175.583,49.934,160.564
C06807=1024.740,440.186,-160.804,175.565,49.930,160.560
C06808=1024.727,439.942,-160.750,175.546,49.926,160.556
C06809=1024.713,439.698,-160.698,175.529,49.922,160.552
C06810=1024.698,439.454,-160.645,175.511,49.918,160.548
C06811=1024.685,439.210,-160.593,175.492,49.915,160.543
C06812=1024.672,438.966,-160.540,175.475,49.911,160.539
C06813=1024.658,438.722,-160.487,175.457,49.907,160.535
C06814=1024.644,438.478,-160.435,175.439,49.903,160.531
C06815=1024.631,438.234,-160.383,175.422,49.899,160.527
C06816=1024.618,437.990,-160.330,175.404,49.896,160.523
C06817=1024.604,437.745,-160.278,175.386,49.892,160.519
C06818=1024.591,437.501,-160.226,175.369,49.888,160.515
C06819=1024.577,437.257,-160.174,175.351,49.885,160.511
C06820=1024.563,437.013,-160.122,175.334,49.881,160.507
C06821=1024.551,436.769,-160.069,175.316,49.877,160.503
C06822=1024.537,436.524,-160.017,175.300,49.873,160.499
C06823=1024.524,436.280,-159.966,175.283,49.870,160.495
C06824=1024.510,436.036,-159.914,175.265,49.866,160.491
C06825=1024.497,435.791,-159.862,175.248,49.862,160.487
C06826=1024.484,435.547,-159.811,175.231,49.859,160.483
C06827=1024.471,435.303,-159.758,175.214,49.855,160.479
C06828=1024.458,435.058,-159.707,175.197,49.852,160.476
C06829=1024.445,434.814,-159.656,175.180,49.848,160.472
C06830=1024.431,434.570,-159.604,175.164,49.844,160.468
C06831=1024.418,434.325,-159.553,175.147,49.841,160.464
C06832=1024.406,434.081,-159.502,175.130,49.838,160.460
C06833=1024.392,433.836,-159.450,175.113,49.834,160.456
C06834=1024.379,433.592,-159.399,175.097,49.831,160.453
C06835=1024.366,433.347,-159.348,175.080,49.827,160.449
C06836=1024.354,433.103,-159.297,175.063,49.824,160.445
C06837=1024.341,432.859,-159.245,175.048,49.820,160.442
C06838=1024.327,432.615,-159.194,175.031,49.816,160.438
C06839=1024.315,432.369,-159.144,175.014,49.813,160.434
C06840=1024.302,432.125,-159.093,174.998,49.810,160.430
C06841=1024.289,431.880,-159.042,174.983,49.807,160.427
C06842=1024.276,431.636,-158.991,174.966,49.804,160.423
C06843=1024.264,431.391,-158.941,174.950,49.800,160.419
C06844=1024.251,431.147,-158.890,174.934,49.797,160.416
C06845=1024.238,430.902,-158.839,174.918,49.793,160.412
C06846=1024.226,430.657,-158.789,174.902,49.791,160.409
C06847=1024.213,430.413,-158.738,174.886,49.787,160.405
C06848=1024.200,430.168,-158.689,174.870,49.784,160.402
C06849=1024.187,429.924,-158.638,174.854,49.781,160.398
C06850=1024.175,429.679,-158.588,174.838,49.777,160.394
C06851=1024.163,429.435,-158.538,174.823,49.775,160.391
C06852=1024.150,429.190,-158.488,174.807,49.771,160.387
C06853=1024.138,428.946,-158.437,174.792,49.768,160.384
C06854=1024.125,428.701,-158.387,174.776,49.765,160.381
C06855=1024.113,428.456,-158.337,174.760,49.762,160.377
C06856=1024.101,428.211,-158.287,174.745,49.759,160.374
C06857=1024.088,427.967,-158.237,174.730,49.756,160.370
C06858=1024.075,427.722,-158.187,174.715,49.753,160.367
C06859=1024.063,427.477,-158.137,174.699,49.750,160.364
C06860=1024.051,427.233,-158.087,174.684,49.747,160.360
C06861=1024.039,426.987,-158.038,174.669,49.743,160.357
C06862=1024.022,426.652,-157.969,174.648,49.740,160.352
C06863=1024.005,426.316,-157.901,174.627,49.735,160.348
C06864=1023.990,425.981,-157.833,174.607,49.731,160.343
C06865=1023.973,425.645,-157.765,174.586,49.727,160.338
C06866=1023.961,425.401,-157.716,174.572,49.724,160.335
C06867=1023.949,425.156,-157.667,174.556,49.721,160.332
C06868=1023.937,424.910,-157.617,174.542,49.719,160.329
C06869=1023.925,424.666,-157.569,174.527,49.716,160.325
C06870=1023.912,424.421,-157.519,174.513,49.713,160.322
C06871=1023.901,424.176,-157.470,174.497,49.711,160.319
C06872=1023.888,423.931,-157.421,174.483,49.707,160.316
C06873=1023.877,423.686,-157.372,174.468,49.705,160.313
C06874=1023.865,423.442,-157.323,174.454,49.702,160.310
C06875=1023.853,423.197,-157.274,174.440,49.699,160.307
C06876=1023.841,422.952,-157.225,174.425,49.697,160.303
C06877=1023.830,422.706,-157.177,174.410,49.694,160.300
C06878=1023.817,422.461,-157.128,174.396,49.691,160.297
C06879=1023.806,422.217,-157.079,174.382,49.688,160.294
C06880=1023.795,421.972,-157.030,174.367,49.686,160.291
C06881=1023.783,421.727,-156.982,174.353,49.683,160.288
C06882=1023.771,421.481,-156.933,174.339,49.680,160.285
C06883=1023.759,421.236,-156.885,174.325,49.678,160.282
C06884=1023.747,420.992,-156.836,174.311,49.675,160.279
C06885=1023.736,420.746,-156.789,174.297,49.672,160.276
C06886=1023.724,420.500,-156.740,174.282,49.670,160.273
C06887=1023.712,420.256,-156.692,174.268,49.667,160.270
C06888=1023.701,420.011,-156.643,174.254,49.665,160.267
C06889=1023.689,419.766,-156.596,174.241,49.663,160.264
C06890=1023.678,419.520,-156.547,174.227,49.660,160.261
C06891=1023.666,419.275,-156.500,174.213,49.658,160.258
C06892=1023.655,419.030,-156.451,174.199,49.655,160.255
C06893=1023.643,418.785,-156.404,174.185,49.653,160.252
C06894=1023.632,418.540,-156.356,174.172,49.650,160.249
C06895=1023.621,418.295,-156.308,174.158,49.648,160.246
C06896=1023.609,418.050,-156.260,174.145,49.645,160.243
C06897=1023.598,417.805,-156.212,174.131,49.643,160.240
C06898=1023.586,417.560,-156.164,174.117,49.641,160.238
C06899=1023.575,417.314,-156.117,174.104,49.638,160.235
C06900=1023.564,417.069,-156.069,174.091,49.636,160.232
C06901=1023.553,416.824,-156.021,174.077,49.633,160.229
C06902=1023.541,416.578,-155.974,174.063,49.631,160.226
C06903=1023.531,416.334,-155.926,174.050,49.629,160.223
C06904=1023.519,416.088,-155.879,174.037,49.627,160.221
C06905=1023.507,415.843,-155.831,174.024,49.624,160.218
C06906=1023.497,415.598,-155.784,174.010,49.623,160.215
C06907=1023.485,415.352,-155.736,173.998,49.620,160.212
C06908=1023.474,415.107,-155.689,173.984,49.618,160.210
C06909=1023.464,414.861,-155.642,173.971,49.615,160.207
C06910=1023.452,414.616,-155.595,173.958,49.614,160.204
C06911=1023.441,414.371,-155.549,173.944,49.611,160.201
C06912=1023.430,414.125,-155.502,173.932,49.609,160.199
C06913=1023.419,413.880,-155.455,173.919,49.607,160.196
C06914=1023.408,413.634,-155.407,173.906,49.605,160.194
C06915=1023.397,413.389,-155.361,173.893,49.603,160.191
C06916=1023.386,413.144,-155.314,173.880,49.601,160.188
C06917=1023.374,412.899,-155.267,173.868,49.599,160.185
C06918=1023.364,412.654,-155.221,173.855,49.597,160.183
C06919=1023.353,412.408,-155.173,173.842,49.595,160.180
C06920=1023.342,412.162,-155.127,173.829,49.593,160.178
C06921=1023.331,411.917,-155.080,173.817,49.591,160.175
C06922=1023.317,411.593,-155.019,173.800,49.588,160.172
C06923=1023.303,411.268,-154.957,173.783,49.585,160.168
C06924=1023.289,410.945,-154.896,173.767,49.583,160.165
C06925=1023.275,410.620,-154.835,173.750,49.580,160.161
C06926=1023.264,410.375,-154.788,173.738,49.579,160.159
C06927=1023.253,410.129,-154.742,173.725,49.577,160.156
C06928=1023.242,409.884,-154.696,173.712,49.575,160.154
C06929=1023.232,409.639,-154.650,173.701,49.573,160.151
C06930=1023.222,409.393,-154.603,173.688,49.571,160.149
C06931=1023.211,409.147,-154.557,173.676,49.569,160.146
C06932=1023.199,408.901,-154.512,173.664,49.567,160.144
C06933=1023.189,408.656,-154.466,173.651,49.566,160.141
C06934=1023.178,408.410,-154.420,173.639,49.564,160.139
C06935=1023.167,408.165,-154.374,173.627,49.562,160.136
C06936=1023.157,407.919,-154.328,173.615,49.560,160.134
C06937=1023.147,407.674,-154.283,173.603,49.559,160.132
C06938=1023.136,407.428,-154.237,173.591,49.557,160.129
C06939=1023.126,407.183,-154.191,173.579,49.556,160.127
C06940=1023.115,406.937,-154.146,173.567,49.554,160.125
C06941=1023.104,406.691,-154.100,173.555,49.552,160.122
C06942=1023.094,406.446,-154.055,173.542,49.550,160.120
C06943=1023.084,406.200,-154.010,173.531,49.549,160.118
C06944=1023.073,405.955,-153.964,173.519,49.547,160.115
C06945=1023.062,405.709,-153.918,173.507,49.546,160.113
C06946=1023.053,405.464,-153.873,173.495,49.544,160.110
C06947=1023.041,405.218,-153.828,173.483,49.543,160.108
C06948=1023.031,404.972,-153.782,173.471,49.541,160.106
C06949=1023.021,404.727,-153.737,173.460,49.539,160.103
C06950=1023.011,404.481,-153.692,173.448,49.538,160.101
C06951=1023.001,404.235,-153.647,173.437,49.536,160.099
C06952=1022.990,403.990,-153.601,173.425,49.535,160.097
C06953=1022.981,403.744,-153.556,173.413,49.534,160.094
C06954=1022.969,403.498,-153.512,173.402,49.532,160.092
C06955=1022.960,403.253,-153.467,173.390,49.531,160.090
C06956=1022.949,403.007,-153.421,173.378,49.529,160.088
C06957=1022.939,402.762,-153.376,173.367,49.528,160.085
C06958=1022.930,402.516,-153.331,173.356,49.526,160.083
C06959=1022.919,402.270,-153.286,173.344,49.525,160.081
C06960=1022.910,402.025,-153.241,173.332,49.523,160.079
C06961=1022.899,401.779,-153.197,173.322,49.522,160.077
C06962=1022.889,401.533,-153.152,173.310,49.521,160.074
C06963=1022.879,401.288,-153.107,173.299,49.519,160.072
C06964=1022.869,401.042,-153.062,173.288,49.517,160.070
C06965=1022.860,400.796,-153.018,173.276,49.516,160.068
C06966=1022.849,400.550,-152.973,173.265,49.515,160.066
C06967=1022.839,400.305,-152.929,173.254,49.514,160.064
C06968=1022.830,400.058,-152.884,173.242,49.513,160.061
C06969=1022.819,399.813,-152.840,173.232,49.511,160.059
C06970=1022.810,399.568,-152.795,173.220,49.510,160.057
C06971=1022.800,399.322,-152.751,173.209,49.509,160.055
C06972=1022.790,399.076,-152.707,173.198,49.508,160.053
C06973=1022.780,398.830,-152.663,173.187,49.506,160.051
C06974=1022.770,398.583,-152.619,173.176,49.505,160.049
C06975=1022.760,398.338,-152.574,173.166,49.504,160.047
C06976=1022.751,398.092,-152.530,173.154,49.503,160.045
C06977=1022.740,397.846,-152.487,173.143,49.502,160.043
C06978=1022.731,397.601,-152.442,173.133,49.500,160.041
C06979=1022.721,397.355,-152.398,173.122,49.500,160.039
C06980=1022.711,397.109,-152.354,173.111,49.498,160.037
C06981=1022.701,396.863,-152.311,173.100,49.498,160.035
C06982=1022.690,396.562,-152.257,173.087,49.496,160.032
C06983=1022.677,396.260,-152.203,173.074,49.495,160.030
C06984=1022.665,395.957,-152.150,173.061,49.494,160.027
C06985=1022.654,395.656,-152.096,173.047,49.493,160.025
C06986=1022.644,395.410,-152.052,173.036,49.491,160.023
C06987=1022.634,395.164,-152.008,173.026,49.490,160.021
C06988=1022.624,394.918,-151.965,173.015,49.490,160.019
C06989=1022.615,394.673,-151.922,173.005,49.489,160.017
C06990=1022.605,394.426,-151.878,172.994,49.487,160.015
C06991=1022.595,394.181,-151.835,172.984,49.487,160.013
C06992=1022.586,393.934,-151.791,172.973,49.486,160.011
C06993=1022.577,393.689,-151.748,172.962,49.485,160.009
C06994=1022.567,393.443,-151.704,172.952,49.484,160.008
C06995=1022.557,393.196,-151.661,172.942,49.483,160.006
C06996=1022.549,392.951,-151.617,172.931,49.482,160.004
C06997=1022.539,392.704,-151.575,172.921,49.481,160.002
C06998=1022.529,392.459,-151.531,172.910,49.481,160.000
C06999=1022.519,392.213,-151.489,172.900,49.480,159.998
C07000=1022.510,391.966,-151.445,172.890,49.479,159.996
C07001=1022.501,391.721,-151.402,172.880,49.478,159.994
C07002=1022.491,391.474,-151.359,172.869,49.477,159.993
C07003=1022.482,391.229,-151.317,172.859,49.477,159.991
C07004=1022.473,390.982,-151.274,172.849,49.476,159.989
C07005=1022.463,390.736,-151.231,172.839,49.475,159.987
C07006=1022.453,390.490,-151.188,172.828,49.475,159.985
C07007=1022.445,390.244,-151.145,172.818,49.474,159.983
C07008=1022.435,389.998,-151.102,172.808,49.474,159.982
C07009=1022.426,389.752,-151.059,172.798,49.473,159.980
C07010=1022.416,389.506,-151.017,172.787,49.472,159.978
C07011=1022.407,389.260,-150.973,172.778,49.471,159.976
C07012=1022.398,389.014,-150.931,172.767,49.470,159.974
C07013=1022.388,388.767,-150.888,172.758,49.470,159.973
C07014=1022.379,388.521,-150.847,172.747,49.469,159.971
C07015=1022.370,388.275,-150.804,172.737,49.469,159.969
C07016=1022.360,388.029,-150.761,172.729,49.468,159.968
C07017=1022.352,387.783,-150.718,172.718,49.467,159.966
C07018=1022.343,387.536,-150.677,172.709,49.467,159.964
C07019=1022.333,387.290,-150.634,172.699,49.467,159.963
C07020=1022.324,387.044,-150.591,172.689,49.466,159.961
C07021=1022.315,386.798,-150.550,172.679,49.465,159.959
C07022=1022.305,386.552,-150.507,172.669,49.465,159.957
C07023=1022.296,386.305,-150.465,172.659,49.465,159.956
C07024=1022.287,386.059,-150.423,172.649,49.465,159.954
C07025=1022.278,385.813,-150.381,172.639,49.464,159.952
C07026=1022.269,385.567,-150.339,172.630,49.463,159.951
C07027=1022.260,385.321,-150.297,172.620,49.463,159.949
C07028=1022.251,385.075,-150.255,172.610,49.462,159.947
C07029=1022.241,384.827,-150.213,172.601,49.463,159.946
C07030=1022.232,384.581,-150.171,172.591,49.462,159.944
C07031=1022.223,384.335,-150.129,172.581,49.462,159.943
C07032=1022.214,384.089,-150.087,172.572,49.461,159.941
C07033=1022.204,383.843,-150.046,172.563,49.461,159.939
C07034=1022.195,383.597,-150.004,172.553,49.460,159.938
C07035=1022.186,383.350,-149.963,172.543,49.460,159.936
C07036=1022.178,383.104,-149.921,172.534,49.460,159.935
C07037=1022.169,382.857,-149.879,172.525,49.460,159.933
C07038=1022.160,382.611,-149.837,172.515,49.459,159.931
C07039=1022.150,382.365,-149.796,172.505,49.460,159.930
C07040=1022.141,382.119,-149.755,172.496,49.459,159.928
C07041=1022.132,381.872,-149.714,172.486,49.459,159.927
C07042=1022.123,381.608,-149.669,172.477,49.458,159.925
C07043=1022.113,381.343,-149.624,172.467,49.459,159.924
C07044=1022.104,381.078,-149.580,172.456,49.459,159.922
C07045=1022.095,380.814,-149.536,172.446,49.458,159.920
C07046=1022.086,380.567,-149.494,172.437,49.458,159.919
C07047=1022.077,380.320,-149.453,172.428,49.458,159.917
C07048=1022.068,380.074,-149.411,172.419,49.458,159.916
C07049=1022.059,379.828,-149.369,172.410,49.457,159.914
C07050=1022.050,379.582,-149.329,172.400,49.458,159.913
C07051=1022.042,379.335,-149.288,172.390,49.457,159.911
C07052=1022.033,379.088,-149.247,172.382,49.457,159.910
C07053=1022.025,378.843,-149.205,172.373,49.457,159.908
C07054=1022.017,378.628,-149.170,172.365,49.457,159.907
C07055=1022.009,378.414,-149.134,172.357,49.457,159.906
C07056=1022.002,378.200,-149.099,172.349,49.457,159.905
C07057=1021.994,377.986,-149.063,172.341,49.457,159.903
C07058=1021.987,377.772,-149.027,172.333,49.456,159.902
C07059=1021.979,377.558,-148.992,172.325,49.457,159.901
C07060=1021.972,377.343,-148.956,172.318,49.457,159.899
C07061=1021.964,377.130,-148.920,172.310,49.457,159.898
C07062=1021.956,376.883,-148.879,172.301,49.457,159.897
C07063=1021.948,376.636,-148.838,172.292,49.457,159.896
C07064=1021.939,376.390,-148.798,172.283,49.457,159.894
C07065=1021.930,376.143,-148.757,172.274,49.457,159.893
C07066=1021.921,375.897,-148.717,172.265,49.457,159.891
C07067=1021.913,375.650,-148.676,172.256,49.457,159.890
C07068=1021.904,375.405,-148.636,172.247,49.457,159.889
C07069=1021.895,375.158,-148.595,172.238,49.458,159.887
C07070=1021.887,374.912,-148.555,172.229,49.457,159.886
C07071=1021.878,374.665,-148.514,172.220,49.458,159.884
C07072=1021.869,374.419,-148.474,172.212,49.458,159.883
C07073=1021.861,374.171,-148.434,172.203,49.458,159.882
C07074=1021.852,373.925,-148.394,172.194,49.458,159.880
C07075=1021.843,373.678,-148.353,172.186,49.459,159.879
C07076=1021.835,373.432,-148.313,172.176,49.459,159.878
C07077=1021.827,373.185,-148.273,172.168,49.459,159.876
C07078=1021.818,372.938,-148.232,172.160,49.459,159.875
C07079=1021.810,372.692,-148.192,172.150,49.460,159.874
C07080=1021.801,372.446,-148.152,172.142,49.460,159.873
C07081=1021.793,372.199,-148.111,172.134,49.460,159.871
C07082=1021.784,371.952,-148.072,172.125,49.461,159.870
C07083=1021.776,371.706,-148.031,172.116,49.461,159.869
C07084=1021.768,371.459,-147.992,172.108,49.461,159.867
C07085=1021.759,371.212,-147.951,172.098,49.462,159.866
C07086=1021.750,370.966,-147.912,172.090,49.462,159.865
C07087=1021.742,370.719,-147.871,172.082,49.463,159.864
C07088=1021.734,370.473,-147.832,172.074,49.462,159.862
C07089=1021.726,370.226,-147.792,172.065,49.463,159.861
C07090=1021.717,369.979,-147.752,172.056,49.463,159.860
C07091=1021.709,369.732,-147.712,172.048,49.464,159.858
C07092=1021.701,369.486,-147.672,172.040,49.464,159.857
C07093=1021.693,369.239,-147.632,172.031,49.465,159.856
C07094=1021.684,368.993,-147.592,172.022,49.465,159.855
C07095=1021.677,368.746,-147.552,172.014,49.465,159.854
C07096=1021.668,368.499,-147.513,172.006,49.466,159.852
C07097=1021.660,368.252,-147.473,171.998,49.466,159.851
C07098=1021.652,368.006,-147.434,171.989,49.467,159.850
C07099=1021.643,367.759,-147.395,171.981,49.468,159.849
C07100=1021.636,367.512,-147.355,171.973,49.468,159.848
C07101=1021.627,367.266,-147.315,171.965,49.469,159.846
C07102=1021.616,366.957,-147.266,171.954,49.469,159.845
C07103=1021.606,366.650,-147.217,171.944,49.470,159.843
C07104=1021.596,366.342,-147.168,171.933,49.471,159.842
C07105=1021.585,366.035,-147.119,171.923,49.471,159.841
C07106=1021.577,365.788,-147.080,171.915,49.472,159.839
C07107=1021.569,365.541,-147.041,171.907,49.473,159.838
C07108=1021.561,365.295,-147.002,171.899,49.473,159.837
C07109=1021.553,365.048,-146.962,171.890,49.474,159.836
C07110=1021.545,364.801,-146.924,171.882,49.475,159.835
C07111=1021.536,364.555,-146.885,171.874,49.476,159.834
C07112=1021.528,364.308,-146.845,171.866,49.476,159.833
C07113=1021.520,364.061,-146.807,171.858,49.477,159.832
C07114=1021.512,363.814,-146.767,171.850,49.478,159.831
C07115=1021.504,363.567,-146.728,171.842,49.478,159.829
C07116=1021.496,363.321,-146.689,171.834,49.479,159.828
C07117=1021.488,363.074,-146.650,171.826,49.480,159.827
C07118=1021.480,362.826,-146.612,171.818,49.480,159.826
C07119=1021.472,362.580,-146.573,171.810,49.481,159.825
C07120=1021.464,362.333,-146.534,171.802,49.482,159.824
C07121=1021.456,362.086,-146.494,171.794,49.482,159.823
C07122=1021.448,361.839,-146.456,171.786,49.483,159.822
C07123=1021.440,361.593,-146.418,171.778,49.484,159.821
C07124=1021.432,361.346,-146.378,171.770,49.485,159.820
C07125=1021.424,361.099,-146.340,171.763,49.486,159.819
C07126=1021.416,360.852,-146.301,171.754,49.487,159.818
C07127=1021.408,360.605,-146.263,171.747,49.488,159.817
C07128=1021.401,360.358,-146.224,171.739,49.488,159.816
C07129=1021.393,360.112,-146.185,171.731,49.489,159.815
C07130=1021.385,359.864,-146.146,171.723,49.490,159.814
C07131=1021.377,359.618,-146.108,171.715,49.491,159.813
C07132=1021.369,359.371,-146.069,171.707,49.492,159.812
C07133=1021.361,359.124,-146.031,171.699,49.493,159.811
C07134=1021.353,358.877,-145.992,171.692,49.494,159.810
C07135=1021.345,358.629,-145.955,171.684,49.495,159.809
C07136=1021.337,358.383,-145.917,171.676,49.496,159.808
C07137=1021.329,358.136,-145.878,171.668,49.497,159.807
C07138=1021.321,357.889,-145.840,171.660,49.498,159.806
C07139=1021.313,357.642,-145.801,171.653,49.499,159.805
C07140=1021.306,357.395,-145.763,171.645,49.500,159.804
C07141=1021.298,357.148,-145.725,171.637,49.501,159.803
C07142=1021.289,356.901,-145.687,171.629,49.502,159.802
C07143=1021.282,356.655,-145.649,171.622,49.503,159.801
C07144=1021.274,356.407,-145.611,171.615,49.504,159.800
C07145=1021.267,356.161,-145.573,171.607,49.506,159.799
C07146=1021.258,355.913,-145.535,171.600,49.507,159.798
C07147=1021.251,355.666,-145.497,171.592,49.508,159.797
C07148=1021.242,355.419,-145.459,171.584,49.509,159.796
C07149=1021.235,355.172,-145.421,171.576,49.510,159.795
C07150=1021.227,354.926,-145.383,171.569,49.511,159.794
C07151=1021.220,354.678,-145.345,171.561,49.512,159.793
C07152=1021.212,354.431,-145.307,171.555,49.513,159.793
C07153=1021.204,354.184,-145.270,171.547,49.515,159.792
C07154=1021.196,353.938,-145.232,171.539,49.516,159.791
C07155=1021.189,353.690,-145.194,171.531,49.517,159.790
C07156=1021.181,353.443,-145.157,171.524,49.518,159.789
C07157=1021.173,353.196,-145.120,171.516,49.519,159.788
C07158=1021.165,352.955,-145.082,171.510,49.521,159.787
C07159=1021.158,352.714,-145.045,171.502,49.522,159.786
C07160=1021.150,352.473,-145.009,171.494,49.523,159.785
